% RSLogix 500 project BINSCRUBBER T SERIES WITH PALLET WASH AND STACKER_WITH_BIN_CALL_BAK721_eulises.RSS, saved by version 11.00.00.00 %
PROJECT "JBT BIN"    % processor: MicroLogix 1400 %

PROGRAM FILES
  LAD 2 "MAIN"  11 rungs
  LAD 3 "START_UP"  22 rungs
  LAD 4 "ENCODER"  11 rungs
  LAD 5 "CRADLE"  26 rungs
  LAD 6 "BRUSH"  53 rungs
  LAD 7 "TANK"  20 rungs
  LAD 8 "AUXILARY"  13 rungs
  LAD 9 "FAULTS"  37 rungs
  LAD 10 "PID ANALOG"  33 rungs  % Scaling %
  LAD 11 "BIN SIZING"  15 rungs  % Bin sizing Pallet, 26", Tall %
  LAD 12 "STACKER"  50 rungs

DATA FILES
  O0 OUTPUT  9 elements
  I1 INPUT  19 elements
  S2 STATUS  66 elements
  B3 BINARY  10 elements
  T4 TIMER  43 elements
  C5 COUNTER  1 elements
  R6 CONTROL  1 elements
  N7 INTEGER  62 elements
  F8 FLOAT  10 elements
  L9   1 elements
  L10   2 elements
  PD11   2 elements

LADDER 2 "MAIN"
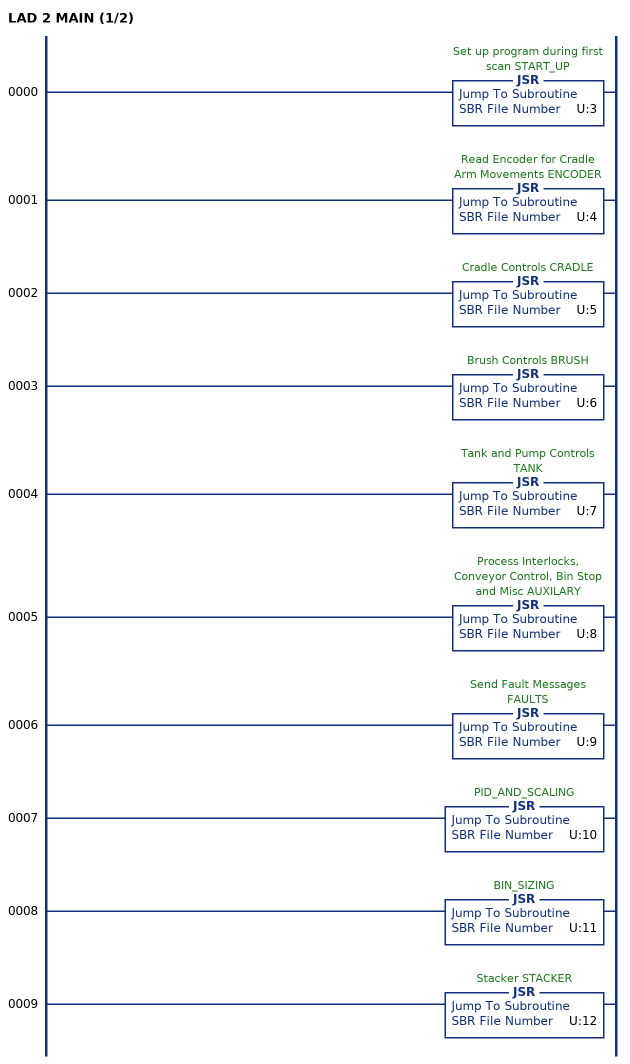
% Rung: 0 %
SOR JSR U:3 EOR
%   U:3  START_UP  "Set up program during first scan" %
% Rung: 1 %
SOR JSR U:4 EOR
%   U:4  ENCODER  "Read Encoder for Cradle Arm Movements" %
% Rung: 2 %
SOR JSR U:5 EOR
%   U:5  CRADLE  "Cradle Controls" %
% Rung: 3 %
SOR JSR U:6 EOR
%   U:6  BRUSH  "Brush Controls" %
% Rung: 4 %
SOR JSR U:7 EOR
%   U:7  TANK  "Tank and Pump Controls" %
% Rung: 5 %
SOR JSR U:8 EOR
%   U:8  AUXILARY  "Process Interlocks, Conveyor Control, Bin Stop and Misc" %
% Rung: 6 %
SOR JSR U:9 EOR
%   U:9  FAULTS  "Send Fault Messages" %
% Rung: 7 %
SOR JSR U:10 EOR
%   U:10  PID_AND_SCALING %
% Rung: 8 %
SOR JSR U:11 EOR
%   U:11  BIN_SIZING %
% Rung: 9 %
SOR JSR U:12 EOR
%   U:12  STACKER  "Stacker" %

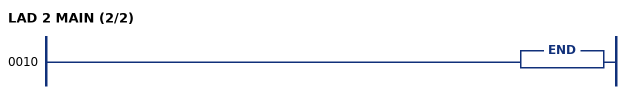
% Rung: 10 %
SOR END EOR

LADDER 3 "START_UP"
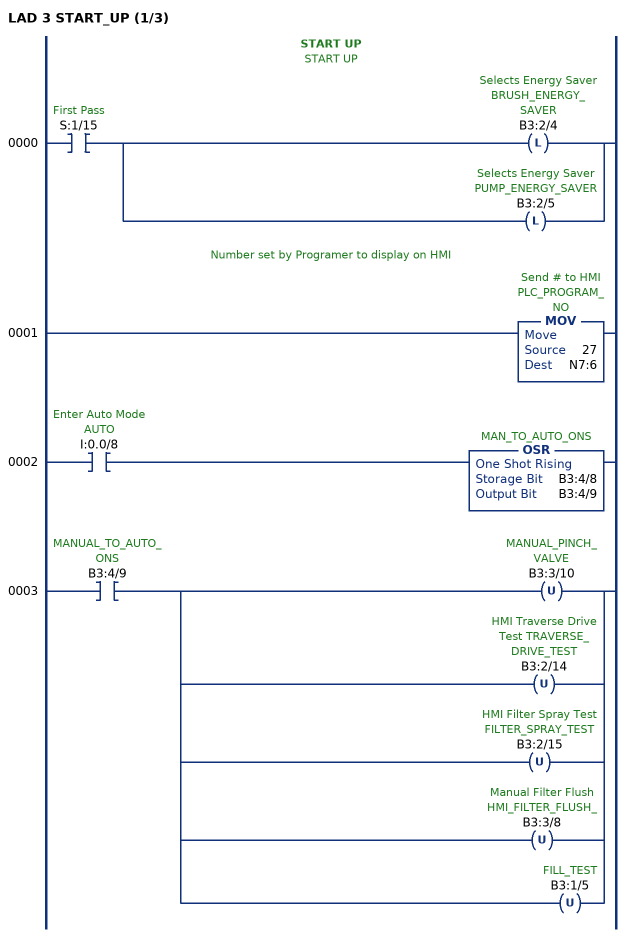
% Rung: 0 %
% TITLE: START UP %
% START UP %
SOR XIC S:1/15 BST OTL B3:2/4 NXB OTL B3:2/5 BND EOR
%   S:1/15  "First Pass" %
%   B3:2/4  BRUSH_ENERGY_SAVER  "Selects Energy Saver" %
%   B3:2/5  PUMP_ENERGY_SAVER  "Selects Energy Saver" %
% Rung: 1 %
% Number set by Programer to display on HMI %
SOR MOV 27 N7:6 EOR
%   N7:6  PLC_PROGRAM_NO  "Send # to HMI" %
% Rung: 2 %
SOR XIC I:0.0/8 OSR B3:4/8 B3:4/9 EOR
%   I:0.0/8  AUTO  "Enter Auto Mode" %
%   B3:4/8  MAN_TO_AUTO_ONS %
%   B3:4/9  MANUAL_TO_AUTO_ONS %
% Rung: 3 %
SOR XIC B3:4/9 BST OTU B3:3/10 NXB BST OTU B3:2/14 NXB BST OTU B3:2/15 NXB BST OTU B3:3/8 NXB OTU B3:1/5 BND BND BND BND EOR
%   B3:4/9  MANUAL_TO_AUTO_ONS %
%   B3:3/10  MANUAL_PINCH_VALVE %
%   B3:2/14  TRAVERSE_DRIVE_TEST  "HMI Traverse Drive Test" %
%   B3:2/15  FILTER_SPRAY_TEST  "HMI Filter Spray Test" %
%   B3:3/8  HMI_FILTER_FLUSH_  "Manual Filter Flush" %
%   B3:1/5  FILL_TEST %

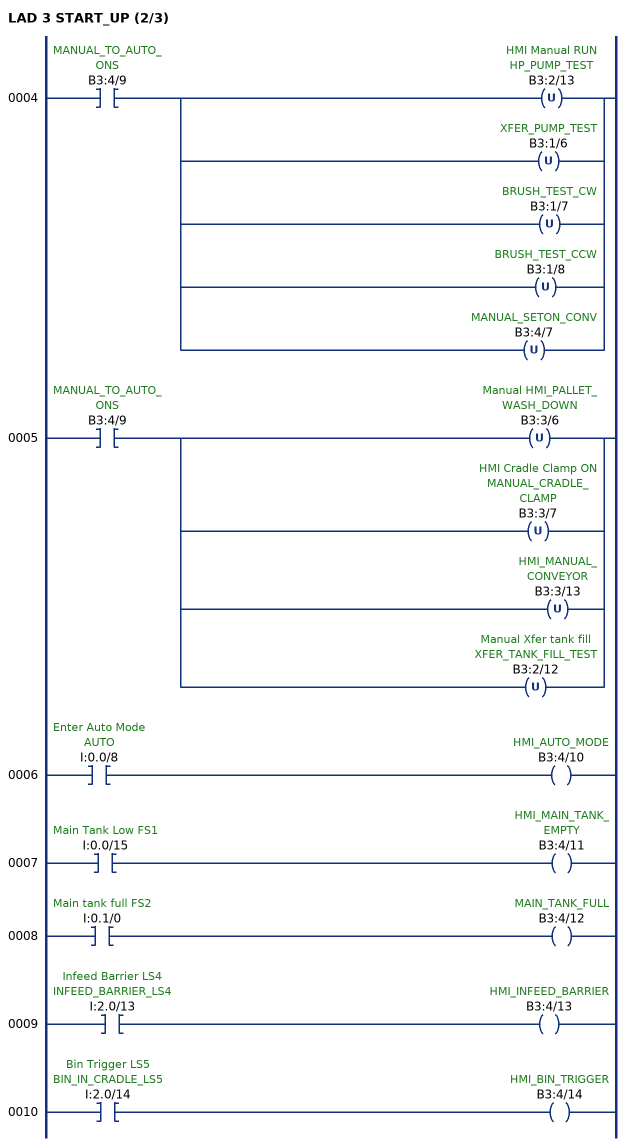
% Rung: 4 %
SOR XIC B3:4/9 BST OTU B3:2/13 NXB BST OTU B3:1/6 NXB BST OTU B3:1/7 NXB BST OTU B3:1/8 NXB OTU B3:4/7 BND BND BND BND EOR
%   B3:4/9  MANUAL_TO_AUTO_ONS %
%   B3:2/13  HP_PUMP_TEST  "HMI Manual RUN" %
%   B3:1/6  XFER_PUMP_TEST %
%   B3:1/7  BRUSH_TEST_CW %
%   B3:1/8  BRUSH_TEST_CCW %
%   B3:4/7  MANUAL_SETON_CONV %
% Rung: 5 %
SOR XIC B3:4/9 BST OTU B3:3/6 NXB BST OTU B3:3/7 NXB BST OTU B3:3/13 NXB OTU B3:2/12 BND BND BND EOR
%   B3:4/9  MANUAL_TO_AUTO_ONS %
%   B3:3/6  HMI_PALLET_WASH_DOWN  "Manual" %
%   B3:3/7  MANUAL_CRADLE_CLAMP  "HMI Cradle Clamp ON" %
%   B3:3/13  HMI_MANUAL_CONVEYOR %
%   B3:2/12  XFER_TANK_FILL_TEST  "Manual Xfer tank fill" %
% Rung: 6 %
SOR XIC I:0.0/8 OTE B3:4/10 EOR
%   I:0.0/8  AUTO  "Enter Auto Mode" %
%   B3:4/10  HMI_AUTO_MODE %
% Rung: 7 %
SOR XIC I:0.0/15 OTE B3:4/11 EOR
%   I:0.0/15  FS1  "Main Tank Low" %
%   B3:4/11  HMI_MAIN_TANK_EMPTY %
% Rung: 8 %
SOR XIC I:0.1/0 OTE B3:4/12 EOR
%   I:0.1/0  FS2  "Main tank full" %
%   B3:4/12  MAIN_TANK_FULL %
% Rung: 9 %
SOR XIC I:2.0/13 OTE B3:4/13 EOR
%   I:2.0/13  INFEED_BARRIER_LS4  "Infeed Barrier LS4" %
%   B3:4/13  HMI_INFEED_BARRIER %
% Rung: 10 %
SOR XIC I:2.0/14 OTE B3:4/14 EOR
%   I:2.0/14  BIN_IN_CRADLE_LS5  "Bin Trigger LS5" %
%   B3:4/14  HMI_BIN_TRIGGER %

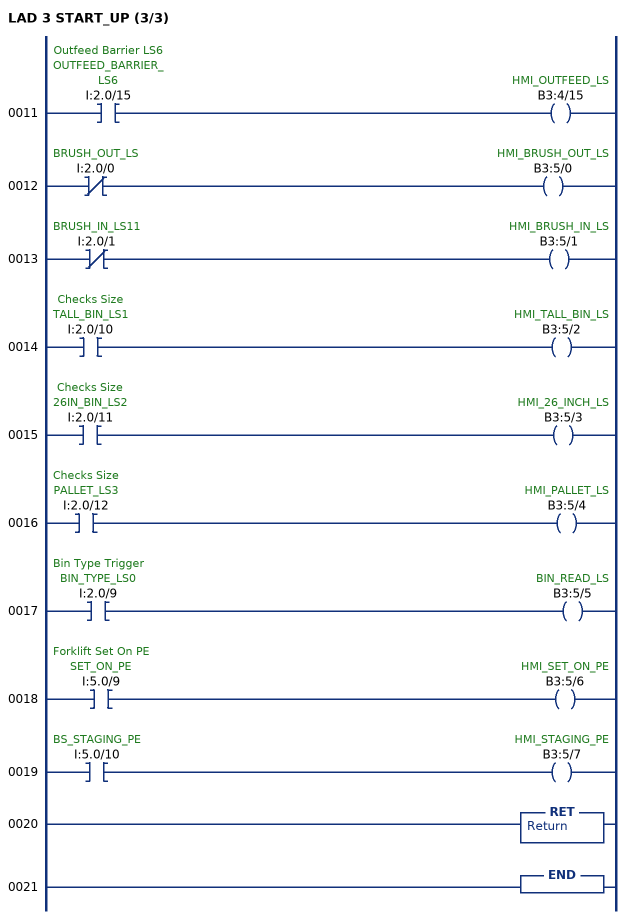
% Rung: 11 %
SOR XIC I:2.0/15 OTE B3:4/15 EOR
%   I:2.0/15  OUTFEED_BARRIER_LS6  "Outfeed Barrier LS6" %
%   B3:4/15  HMI_OUTFEED_LS %
% Rung: 12 %
SOR XIO I:2.0/0 OTE B3:5/0 EOR
%   I:2.0/0  BRUSH_OUT_LS %
%   B3:5/0  HMI_BRUSH_OUT_LS %
% Rung: 13 %
SOR XIO I:2.0/1 OTE B3:5/1 EOR
%   I:2.0/1  BRUSH_IN_LS11 %
%   B3:5/1  HMI_BRUSH_IN_LS %
% Rung: 14 %
SOR XIC I:2.0/10 OTE B3:5/2 EOR
%   I:2.0/10  TALL_BIN_LS1  "Checks Size" %
%   B3:5/2  HMI_TALL_BIN_LS %
% Rung: 15 %
SOR XIC I:2.0/11 OTE B3:5/3 EOR
%   I:2.0/11  26IN_BIN_LS2  "Checks Size" %
%   B3:5/3  HMI_26_INCH_LS %
% Rung: 16 %
SOR XIC I:2.0/12 OTE B3:5/4 EOR
%   I:2.0/12  PALLET_LS3  "Checks Size" %
%   B3:5/4  HMI_PALLET_LS %
% Rung: 17 %
SOR XIC I:2.0/9 OTE B3:5/5 EOR
%   I:2.0/9  BIN_TYPE_LS0  "Bin Type Trigger" %
%   B3:5/5  BIN_READ_LS %
% Rung: 18 %
SOR XIC I:5.0/9 OTE B3:5/6 EOR
%   I:5.0/9  SET_ON_PE  "Forklift Set On PE" %
%   B3:5/6  HMI_SET_ON_PE %
% Rung: 19 %
SOR XIC I:5.0/10 OTE B3:5/7 EOR
%   I:5.0/10  BS_STAGING_PE %
%   B3:5/7  HMI_STAGING_PE %
% Rung: 20 %
SOR RET EOR
% Rung: 21 %
SOR END EOR

LADDER 4 "ENCODER"
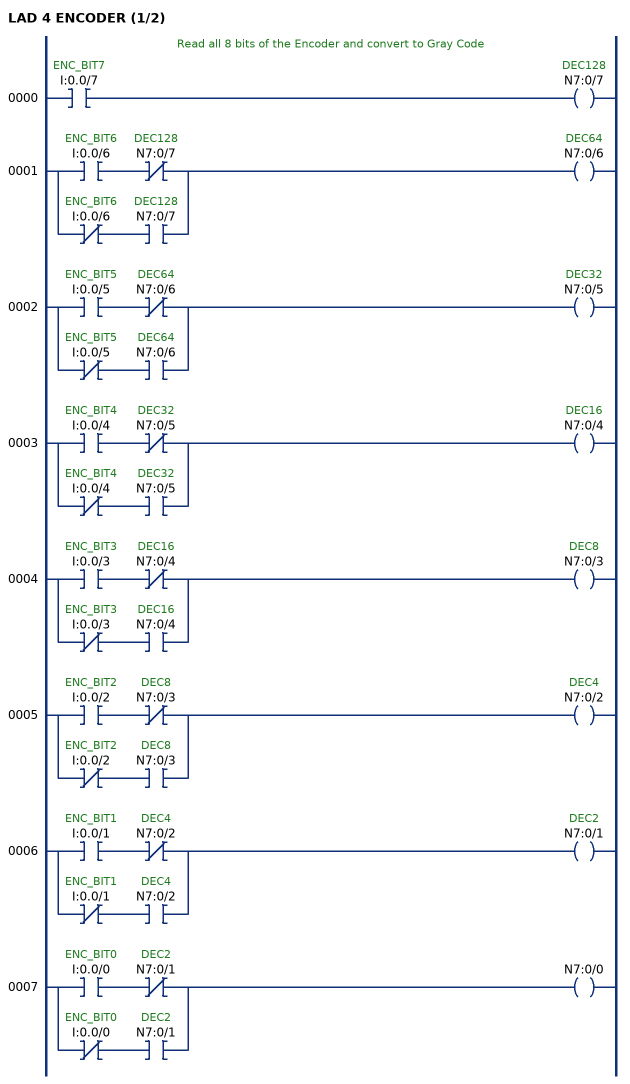
% Rung: 0 %
% Read all 8 bits of the Encoder and convert to Gray Code %
SOR XIC I:0.0/7 OTE N7:0/7 EOR
%   I:0.0/7  ENC_BIT7 %
%   N7:0/7  "DEC128" %
% Rung: 1 %
SOR BST XIC I:0.0/6 XIO N7:0/7 NXB XIO I:0.0/6 XIC N7:0/7 BND OTE N7:0/6 EOR
%   I:0.0/6  ENC_BIT6 %
%   N7:0/7  "DEC128" %
%   N7:0/6  "DEC64" %
% Rung: 2 %
SOR BST XIC I:0.0/5 XIO N7:0/6 NXB XIO I:0.0/5 XIC N7:0/6 BND OTE N7:0/5 EOR
%   I:0.0/5  ENC_BIT5 %
%   N7:0/6  "DEC64" %
%   N7:0/5  "DEC32" %
% Rung: 3 %
SOR BST XIC I:0.0/4 XIO N7:0/5 NXB XIO I:0.0/4 XIC N7:0/5 BND OTE N7:0/4 EOR
%   I:0.0/4  ENC_BIT4 %
%   N7:0/5  "DEC32" %
%   N7:0/4  "DEC16" %
% Rung: 4 %
SOR BST XIC I:0.0/3 XIO N7:0/4 NXB XIO I:0.0/3 XIC N7:0/4 BND OTE N7:0/3 EOR
%   I:0.0/3  ENC_BIT3 %
%   N7:0/4  "DEC16" %
%   N7:0/3  "DEC8" %
% Rung: 5 %
SOR BST XIC I:0.0/2 XIO N7:0/3 NXB XIO I:0.0/2 XIC N7:0/3 BND OTE N7:0/2 EOR
%   I:0.0/2  ENC_BIT2 %
%   N7:0/3  "DEC8" %
%   N7:0/2  "DEC4" %
% Rung: 6 %
SOR BST XIC I:0.0/1 XIO N7:0/2 NXB XIO I:0.0/1 XIC N7:0/2 BND OTE N7:0/1 EOR
%   I:0.0/1  ENC_BIT1 %
%   N7:0/2  "DEC4" %
%   N7:0/1  "DEC2" %
% Rung: 7 %
SOR BST XIC I:0.0/0 XIO N7:0/1 NXB XIO I:0.0/0 XIC N7:0/1 BND OTE N7:0/0 EOR
%   I:0.0/0  ENC_BIT0 %
%   N7:0/1  "DEC2" %

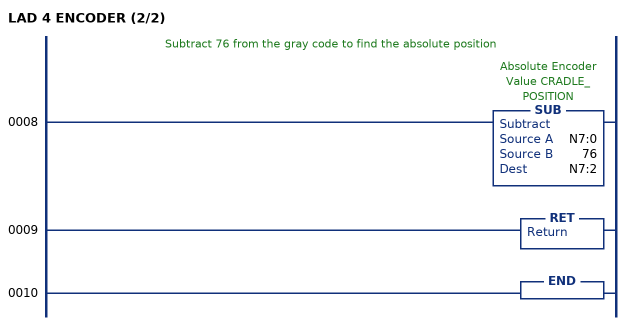
% Rung: 8 %
% Subtract 76 from the gray code to find the absolute position %
SOR SUB N7:0 76 N7:2 EOR
%   N7:0  ENC_POS %
%   N7:2  CRADLE_POSITION  "Absolute Encoder Value" %
% Rung: 9 %
SOR RET EOR
% Rung: 10 %
SOR END EOR

LADDER 5 "CRADLE"
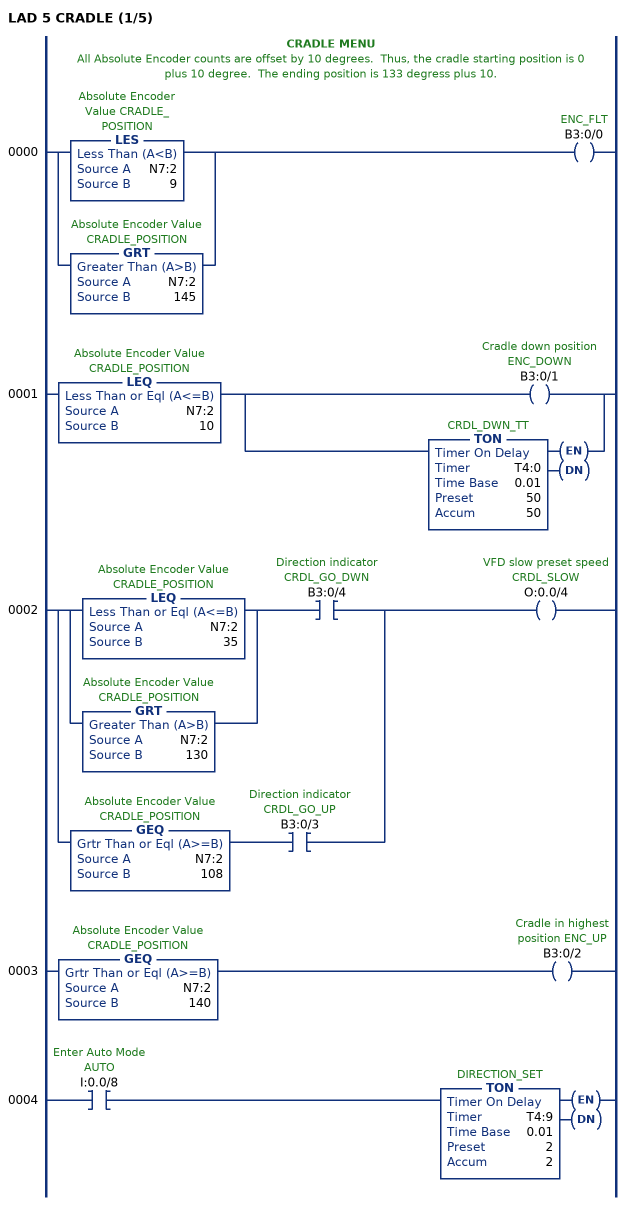
% Rung: 0 %
% TITLE: CRADLE MENU %
% All Absolute Encoder counts are offset by 10 degrees.  Thus, the cradle starting position is 0 plus 10 degree.  The ending position is 133 degress plus 10. %
SOR BST LES N7:2 9 NXB GRT N7:2 145 BND OTE B3:0/0 EOR
%   N7:2  CRADLE_POSITION  "Absolute Encoder Value" %
%   B3:0/0  ENC_FLT %
% Rung: 1 %
SOR LEQ N7:2 10 BST OTE B3:0/1 NXB TON T4:0 0.01 50 50 BND EOR
%   N7:2  CRADLE_POSITION  "Absolute Encoder Value" %
%   B3:0/1  ENC_DOWN  "Cradle down position" %
%   T4:0  CRDL_DWN_TT %
% Rung: 2 %
SOR BST BST LEQ N7:2 35 NXB GRT N7:2 130 BND XIC B3:0/4 NXB GEQ N7:2 108 XIC B3:0/3 BND OTE O:0.0/4 EOR
%   N7:2  CRADLE_POSITION  "Absolute Encoder Value" %
%   B3:0/4  CRDL_GO_DWN  "Direction indicator" %
%   B3:0/3  CRDL_GO_UP  "Direction indicator" %
%   O:0.0/4  CRDL_SLOW  "VFD slow preset speed" %
% Rung: 3 %
SOR GEQ N7:2 140 OTE B3:0/2 EOR
%   N7:2  CRADLE_POSITION  "Absolute Encoder Value" %
%   B3:0/2  ENC_UP  "Cradle in highest position" %
% Rung: 4 %
SOR XIC I:0.0/8 TON T4:9 0.01 2 2 EOR
%   I:0.0/8  AUTO  "Enter Auto Mode" %
%   T4:9  DIRECTION_SET %

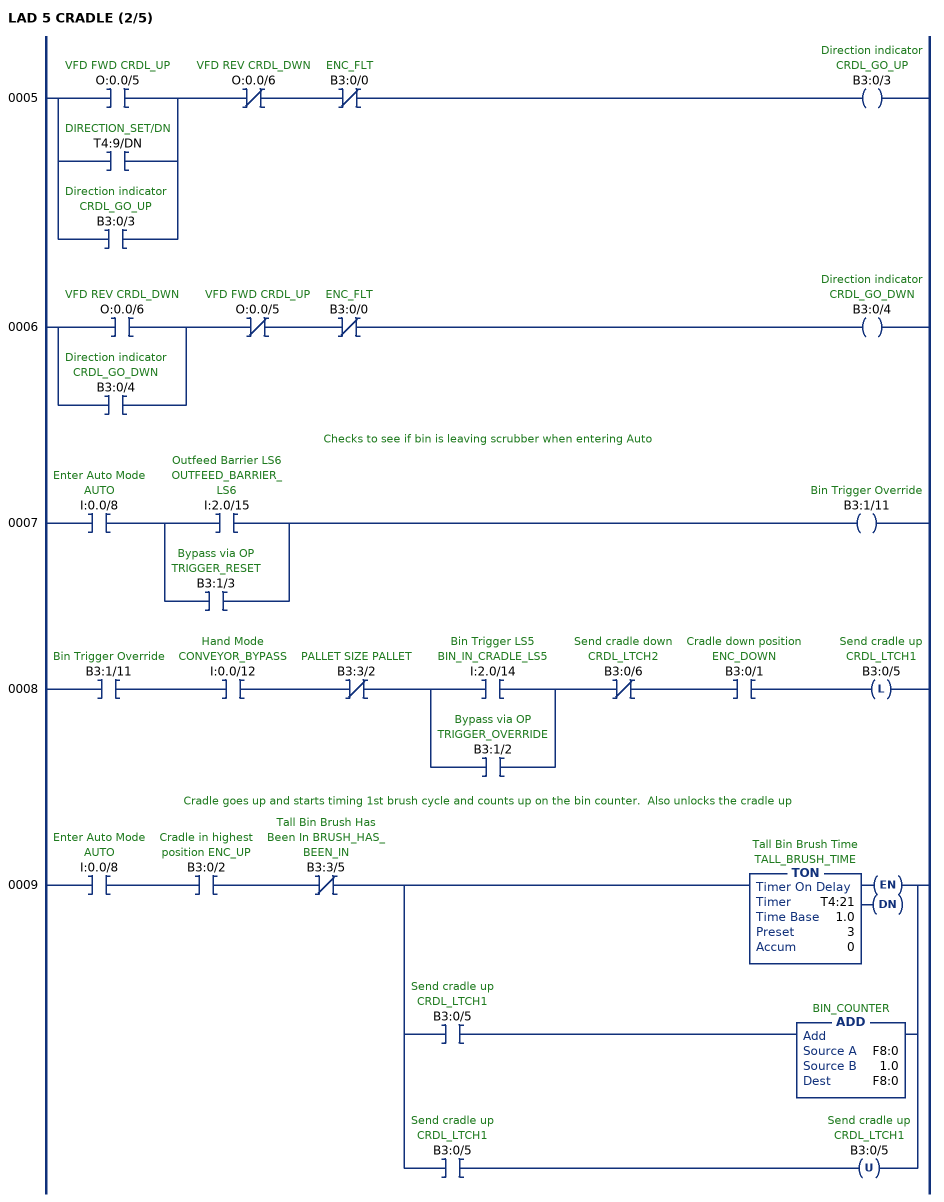
% Rung: 5 %
SOR BST XIC O:0.0/5 NXB XIC T4:9/DN NXB XIC B3:0/3 BND XIO O:0.0/6 XIO B3:0/0 OTE B3:0/3 EOR
%   O:0.0/5  CRDL_UP  "VFD FWD" %
%   T4:9  DIRECTION_SET %
%   B3:0/3  CRDL_GO_UP  "Direction indicator" %
%   O:0.0/6  CRDL_DWN  "VFD REV" %
%   B3:0/0  ENC_FLT %
% Rung: 6 %
SOR BST XIC O:0.0/6 NXB XIC B3:0/4 BND XIO O:0.0/5 XIO B3:0/0 OTE B3:0/4 EOR
%   O:0.0/6  CRDL_DWN  "VFD REV" %
%   B3:0/4  CRDL_GO_DWN  "Direction indicator" %
%   O:0.0/5  CRDL_UP  "VFD FWD" %
%   B3:0/0  ENC_FLT %
% Rung: 7 %
% Checks to see if bin is leaving scrubber when entering Auto %
SOR XIC I:0.0/8 BST XIC I:2.0/15 NXB XIC B3:1/3 BND OTE B3:1/11 EOR
%   I:0.0/8  AUTO  "Enter Auto Mode" %
%   I:2.0/15  OUTFEED_BARRIER_LS6  "Outfeed Barrier LS6" %
%   B3:1/3  TRIGGER_RESET  "Bypass via OP" %
%   B3:1/11  "Bin Trigger Override" %
% Rung: 8 %
SOR XIC B3:1/11 XIC I:0.0/12 XIO B3:3/2 BST XIC I:2.0/14 NXB XIC B3:1/2 BND XIO B3:0/6 XIC B3:0/1 OTL B3:0/5 EOR
%   B3:1/11  "Bin Trigger Override" %
%   I:0.0/12  CONVEYOR_BYPASS  "Hand Mode" %
%   B3:3/2  PALLET  "PALLET SIZE" %
%   I:2.0/14  BIN_IN_CRADLE_LS5  "Bin Trigger LS5" %
%   B3:1/2  TRIGGER_OVERRIDE  "Bypass via OP" %
%   B3:0/6  CRDL_LTCH2  "Send cradle down" %
%   B3:0/1  ENC_DOWN  "Cradle down position" %
%   B3:0/5  CRDL_LTCH1  "Send cradle up" %
% Rung: 9 %
% Cradle goes up and starts timing 1st brush cycle and counts up on the bin counter.  Also unlocks the cradle up %
SOR XIC I:0.0/8 XIC B3:0/2 XIO B3:3/5 BST TON T4:21 1.0 3 0 NXB BST XIC B3:0/5 ADD F8:0 1.0 F8:0 NXB XIC B3:0/5 OTU B3:0/5 BND BND EOR
%   I:0.0/8  AUTO  "Enter Auto Mode" %
%   B3:0/2  ENC_UP  "Cradle in highest position" %
%   B3:3/5  BRUSH_HAS_BEEN_IN  "Tall Bin Brush Has Been In" %
%   T4:21  TALL_BRUSH_TIME  "Tall Bin Brush Time" %
%   B3:0/5  CRDL_LTCH1  "Send cradle up" %
%   F8:0  BIN_COUNTER %

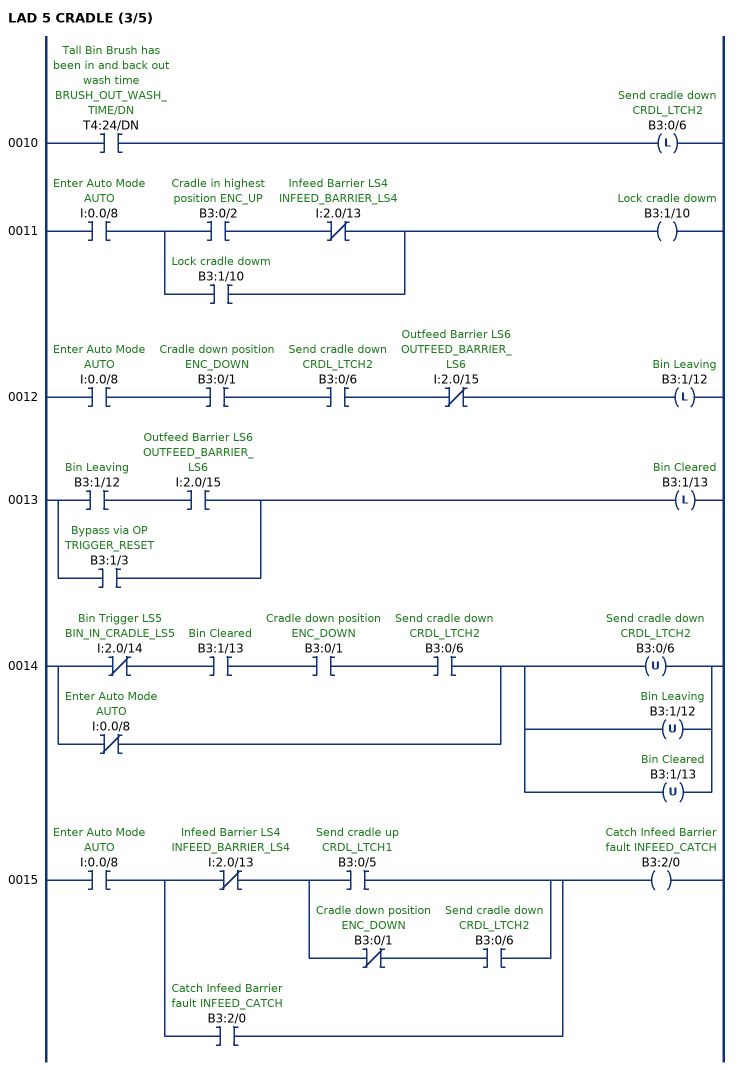
% Rung: 10 %
SOR XIC T4:24/DN OTL B3:0/6 EOR
%   T4:24  BRUSH_OUT_WASH_TIME  "Tall Bin Brush has been in and back out wash time" %
%   B3:0/6  CRDL_LTCH2  "Send cradle down" %
% Rung: 11 %
SOR XIC I:0.0/8 BST XIC B3:0/2 XIO I:2.0/13 NXB XIC B3:1/10 BND OTE B3:1/10 EOR
%   I:0.0/8  AUTO  "Enter Auto Mode" %
%   B3:0/2  ENC_UP  "Cradle in highest position" %
%   I:2.0/13  INFEED_BARRIER_LS4  "Infeed Barrier LS4" %
%   B3:1/10  "Lock cradle dowm" %
% Rung: 12 %
SOR XIC I:0.0/8 XIC B3:0/1 XIC B3:0/6 XIO I:2.0/15 OTL B3:1/12 EOR
%   I:0.0/8  AUTO  "Enter Auto Mode" %
%   B3:0/1  ENC_DOWN  "Cradle down position" %
%   B3:0/6  CRDL_LTCH2  "Send cradle down" %
%   I:2.0/15  OUTFEED_BARRIER_LS6  "Outfeed Barrier LS6" %
%   B3:1/12  "Bin Leaving" %
% Rung: 13 %
SOR BST XIC B3:1/12 XIC I:2.0/15 NXB XIC B3:1/3 BND OTL B3:1/13 EOR
%   B3:1/12  "Bin Leaving" %
%   I:2.0/15  OUTFEED_BARRIER_LS6  "Outfeed Barrier LS6" %
%   B3:1/3  TRIGGER_RESET  "Bypass via OP" %
%   B3:1/13  "Bin Cleared" %
% Rung: 14 %
SOR BST XIO I:2.0/14 XIC B3:1/13 XIC B3:0/1 XIC B3:0/6 NXB XIO I:0.0/8 BND BST OTU B3:0/6 NXB BST OTU B3:1/12 NXB OTU B3:1/13 BND BND EOR
%   I:2.0/14  BIN_IN_CRADLE_LS5  "Bin Trigger LS5" %
%   B3:1/13  "Bin Cleared" %
%   B3:0/1  ENC_DOWN  "Cradle down position" %
%   B3:0/6  CRDL_LTCH2  "Send cradle down" %
%   I:0.0/8  AUTO  "Enter Auto Mode" %
%   B3:1/12  "Bin Leaving" %
% Rung: 15 %
SOR XIC I:0.0/8 BST XIO I:2.0/13 BST XIC B3:0/5 NXB XIO B3:0/1 XIC B3:0/6 BND NXB XIC B3:2/0 BND OTE B3:2/0 EOR
%   I:0.0/8  AUTO  "Enter Auto Mode" %
%   I:2.0/13  INFEED_BARRIER_LS4  "Infeed Barrier LS4" %
%   B3:0/5  CRDL_LTCH1  "Send cradle up" %
%   B3:0/1  ENC_DOWN  "Cradle down position" %
%   B3:0/6  CRDL_LTCH2  "Send cradle down" %
%   B3:2/0  INFEED_CATCH  "Catch Infeed Barrier fault" %

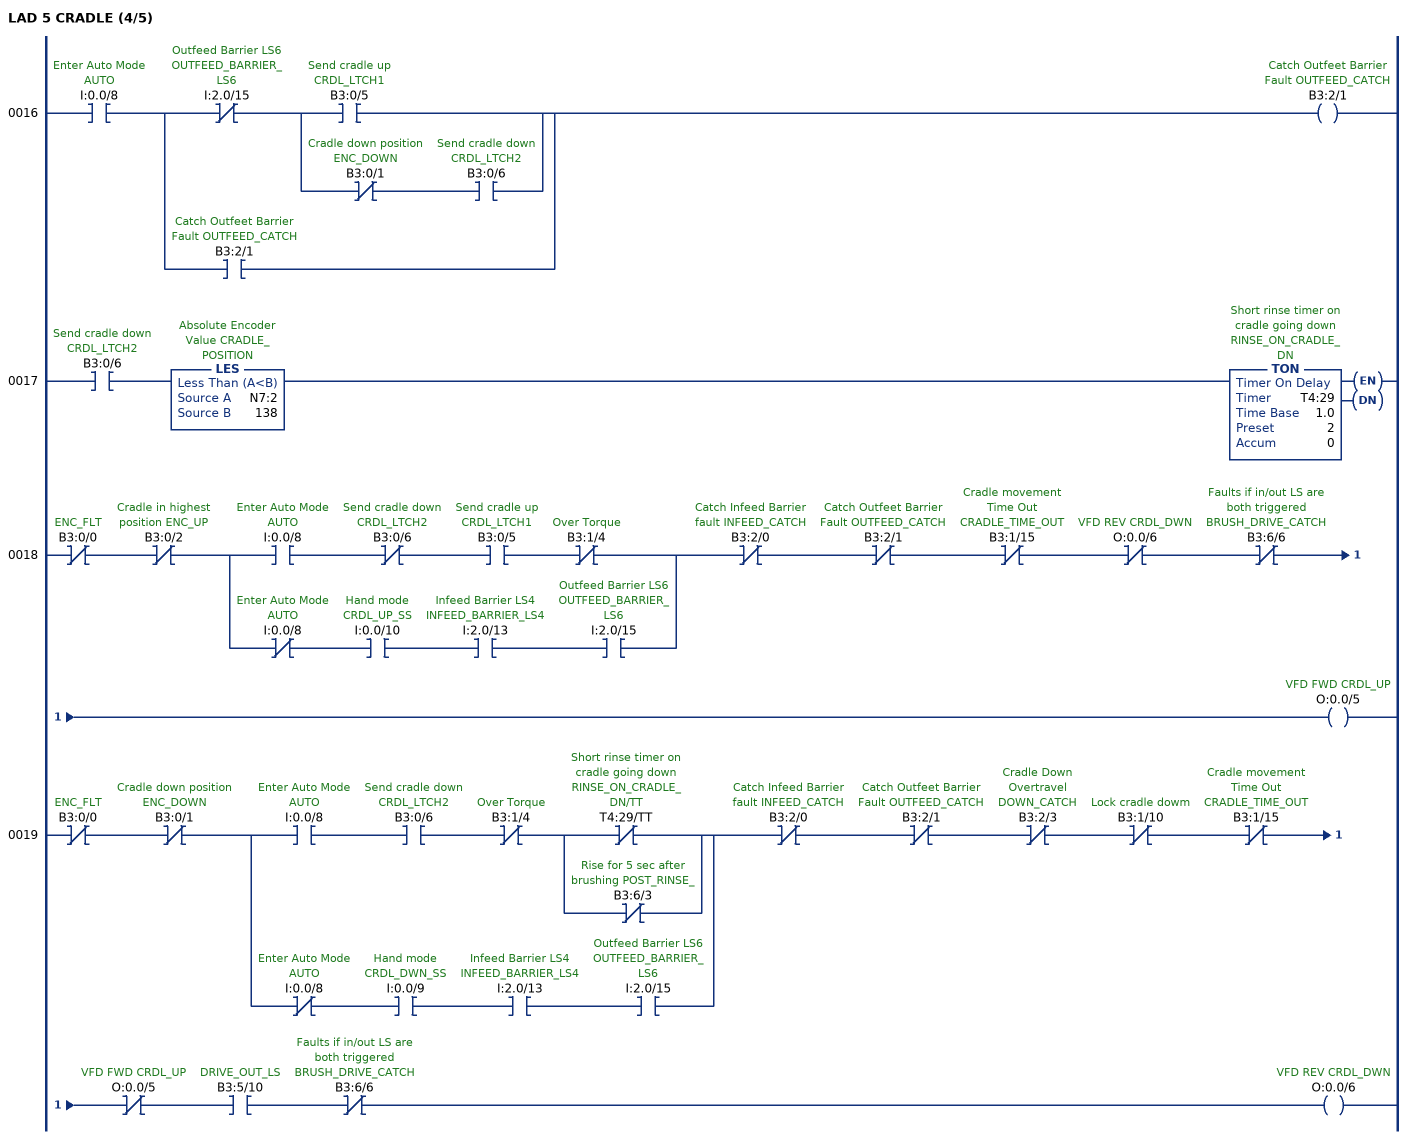
% Rung: 16 %
SOR XIC I:0.0/8 BST XIO I:2.0/15 BST XIC B3:0/5 NXB XIO B3:0/1 XIC B3:0/6 BND NXB XIC B3:2/1 BND OTE B3:2/1 EOR
%   I:0.0/8  AUTO  "Enter Auto Mode" %
%   I:2.0/15  OUTFEED_BARRIER_LS6  "Outfeed Barrier LS6" %
%   B3:0/5  CRDL_LTCH1  "Send cradle up" %
%   B3:0/1  ENC_DOWN  "Cradle down position" %
%   B3:0/6  CRDL_LTCH2  "Send cradle down" %
%   B3:2/1  OUTFEED_CATCH  "Catch Outfeet Barrier Fault" %
% Rung: 17 %
SOR XIC B3:0/6 LES N7:2 138 TON T4:29 1.0 2 0 EOR
%   B3:0/6  CRDL_LTCH2  "Send cradle down" %
%   N7:2  CRADLE_POSITION  "Absolute Encoder Value" %
%   T4:29  RINSE_ON_CRADLE_DN  "Short rinse timer on cradle going down" %
% Rung: 18 %
SOR XIO B3:0/0 XIO B3:0/2 BST XIC I:0.0/8 XIO B3:0/6 XIC B3:0/5 XIO B3:1/4 NXB XIO I:0.0/8 XIC I:0.0/10 XIC I:2.0/13 XIC I:2.0/15 BND XIO B3:2/0 XIO B3:2/1 XIO B3:1/15 XIO O:0.0/6 XIO B3:6/6 OTE O:0.0/5 EOR
%   B3:0/0  ENC_FLT %
%   B3:0/2  ENC_UP  "Cradle in highest position" %
%   I:0.0/8  AUTO  "Enter Auto Mode" %
%   B3:0/6  CRDL_LTCH2  "Send cradle down" %
%   B3:0/5  CRDL_LTCH1  "Send cradle up" %
%   B3:1/4  "Over Torque" %
%   I:0.0/10  CRDL_UP_SS  "Hand mode" %
%   I:2.0/13  INFEED_BARRIER_LS4  "Infeed Barrier LS4" %
%   I:2.0/15  OUTFEED_BARRIER_LS6  "Outfeed Barrier LS6" %
%   B3:2/0  INFEED_CATCH  "Catch Infeed Barrier fault" %
%   B3:2/1  OUTFEED_CATCH  "Catch Outfeet Barrier Fault" %
%   B3:1/15  CRADLE_TIME_OUT  "Cradle movement Time Out" %
%   O:0.0/6  CRDL_DWN  "VFD REV" %
%   B3:6/6  BRUSH_DRIVE_CATCH  "Faults if in/out LS are both triggered" %
%   O:0.0/5  CRDL_UP  "VFD FWD" %
% Rung: 19 %
SOR XIO B3:0/0 XIO B3:0/1 BST XIC I:0.0/8 XIC B3:0/6 XIO B3:1/4 BST XIO T4:29/TT NXB XIO B3:6/3 BND NXB XIO I:0.0/8 XIC I:0.0/9 XIC I:2.0/13 XIC I:2.0/15 BND XIO B3:2/0 XIO B3:2/1 XIO B3:2/3 XIO B3:1/10 XIO B3:1/15 XIO O:0.0/5 XIC B3:5/10 XIO B3:6/6 OTE O:0.0/6 EOR
%   B3:0/0  ENC_FLT %
%   B3:0/1  ENC_DOWN  "Cradle down position" %
%   I:0.0/8  AUTO  "Enter Auto Mode" %
%   B3:0/6  CRDL_LTCH2  "Send cradle down" %
%   B3:1/4  "Over Torque" %
%   T4:29  RINSE_ON_CRADLE_DN  "Short rinse timer on cradle going down" %
%   B3:6/3  POST_RINSE_  "Rise for 5 sec after brushing" %
%   I:0.0/9  CRDL_DWN_SS  "Hand mode" %
%   I:2.0/13  INFEED_BARRIER_LS4  "Infeed Barrier LS4" %
%   I:2.0/15  OUTFEED_BARRIER_LS6  "Outfeed Barrier LS6" %
%   B3:2/0  INFEED_CATCH  "Catch Infeed Barrier fault" %
%   B3:2/1  OUTFEED_CATCH  "Catch Outfeet Barrier Fault" %
%   B3:2/3  DOWN_CATCH  "Cradle Down Overtravel" %
%   B3:1/10  "Lock cradle dowm" %
%   B3:1/15  CRADLE_TIME_OUT  "Cradle movement Time Out" %
%   O:0.0/5  CRDL_UP  "VFD FWD" %
%   B3:5/10  DRIVE_OUT_LS %
%   B3:6/6  BRUSH_DRIVE_CATCH  "Faults if in/out LS are both triggered" %
%   O:0.0/6  CRDL_DWN  "VFD REV" %

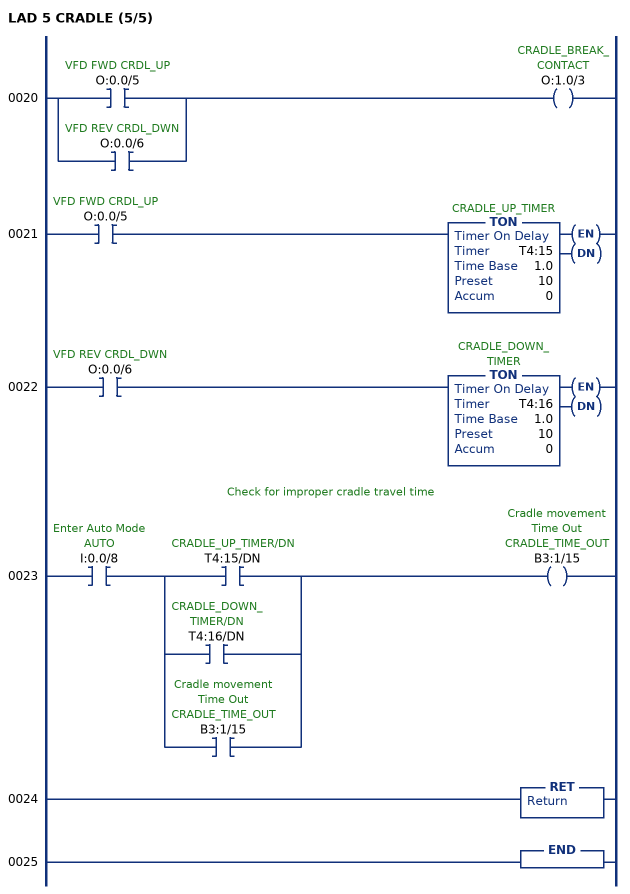
% Rung: 20 %
SOR BST XIC O:0.0/5 NXB XIC O:0.0/6 BND OTE O:1.0/3 EOR
%   O:0.0/5  CRDL_UP  "VFD FWD" %
%   O:0.0/6  CRDL_DWN  "VFD REV" %
%   O:1.0/3  CRADLE_BREAK_CONTACT %
% Rung: 21 %
SOR XIC O:0.0/5 TON T4:15 1.0 10 0 EOR
%   O:0.0/5  CRDL_UP  "VFD FWD" %
%   T4:15  CRADLE_UP_TIMER %
% Rung: 22 %
SOR XIC O:0.0/6 TON T4:16 1.0 10 0 EOR
%   O:0.0/6  CRDL_DWN  "VFD REV" %
%   T4:16  CRADLE_DOWN_TIMER %
% Rung: 23 %
% Check for improper cradle travel time %
SOR XIC I:0.0/8 BST BST XIC T4:15/DN NXB XIC T4:16/DN BND NXB XIC B3:1/15 BND OTE B3:1/15 EOR
%   I:0.0/8  AUTO  "Enter Auto Mode" %
%   T4:15  CRADLE_UP_TIMER %
%   T4:16  CRADLE_DOWN_TIMER %
%   B3:1/15  CRADLE_TIME_OUT  "Cradle movement Time Out" %
% Rung: 24 %
SOR RET EOR
% Rung: 25 %
SOR END EOR

LADDER 6 "BRUSH"
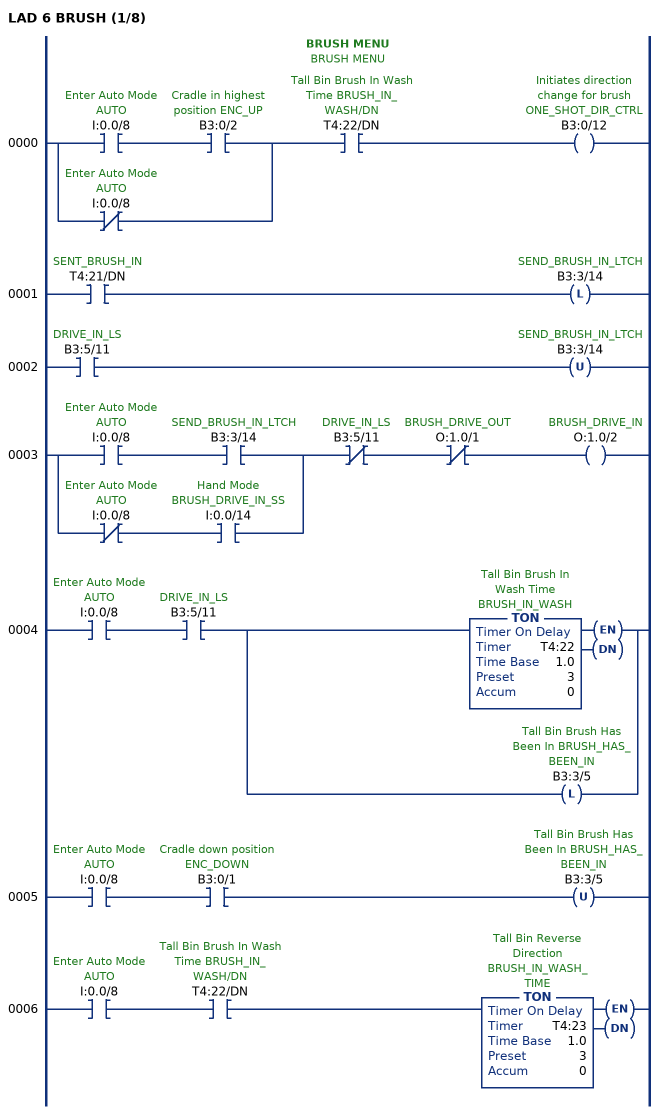
% Rung: 0 %
% TITLE: BRUSH MENU %
% BRUSH MENU %
SOR BST XIC I:0.0/8 XIC B3:0/2 NXB XIO I:0.0/8 BND XIC T4:22/DN OTE B3:0/12 EOR
%   I:0.0/8  AUTO  "Enter Auto Mode" %
%   B3:0/2  ENC_UP  "Cradle in highest position" %
%   T4:22  BRUSH_IN_WASH  "Tall Bin Brush In Wash Time" %
%   B3:0/12  ONE_SHOT_DIR_CTRL  "Initiates direction change for brush" %
% Rung: 1 %
SOR XIC T4:21/DN OTL B3:3/14 EOR
%   T4:21/DN  SENT_BRUSH_IN %
%   B3:3/14  SEND_BRUSH_IN_LTCH %
% Rung: 2 %
SOR XIC B3:5/11 OTU B3:3/14 EOR
%   B3:5/11  DRIVE_IN_LS %
%   B3:3/14  SEND_BRUSH_IN_LTCH %
% Rung: 3 %
SOR BST XIC I:0.0/8 XIC B3:3/14 NXB XIO I:0.0/8 XIC I:0.0/14 BND XIO B3:5/11 XIO O:1.0/1 OTE O:1.0/2 EOR
%   I:0.0/8  AUTO  "Enter Auto Mode" %
%   B3:3/14  SEND_BRUSH_IN_LTCH %
%   I:0.0/14  BRUSH_DRIVE_IN_SS  "Hand Mode" %
%   B3:5/11  DRIVE_IN_LS %
%   O:1.0/1  BRUSH_DRIVE_OUT %
%   O:1.0/2  BRUSH_DRIVE_IN %
% Rung: 4 %
SOR XIC I:0.0/8 XIC B3:5/11 BST TON T4:22 1.0 3 0 NXB OTL B3:3/5 BND EOR
%   I:0.0/8  AUTO  "Enter Auto Mode" %
%   B3:5/11  DRIVE_IN_LS %
%   T4:22  BRUSH_IN_WASH  "Tall Bin Brush In Wash Time" %
%   B3:3/5  BRUSH_HAS_BEEN_IN  "Tall Bin Brush Has Been In" %
% Rung: 5 %
SOR XIC I:0.0/8 XIC B3:0/1 OTU B3:3/5 EOR
%   I:0.0/8  AUTO  "Enter Auto Mode" %
%   B3:0/1  ENC_DOWN  "Cradle down position" %
%   B3:3/5  BRUSH_HAS_BEEN_IN  "Tall Bin Brush Has Been In" %
% Rung: 6 %
SOR XIC I:0.0/8 XIC T4:22/DN TON T4:23 1.0 3 0 EOR
%   I:0.0/8  AUTO  "Enter Auto Mode" %
%   T4:22  BRUSH_IN_WASH  "Tall Bin Brush In Wash Time" %
%   T4:23  BRUSH_IN_WASH_TIME  "Tall Bin Reverse Direction" %

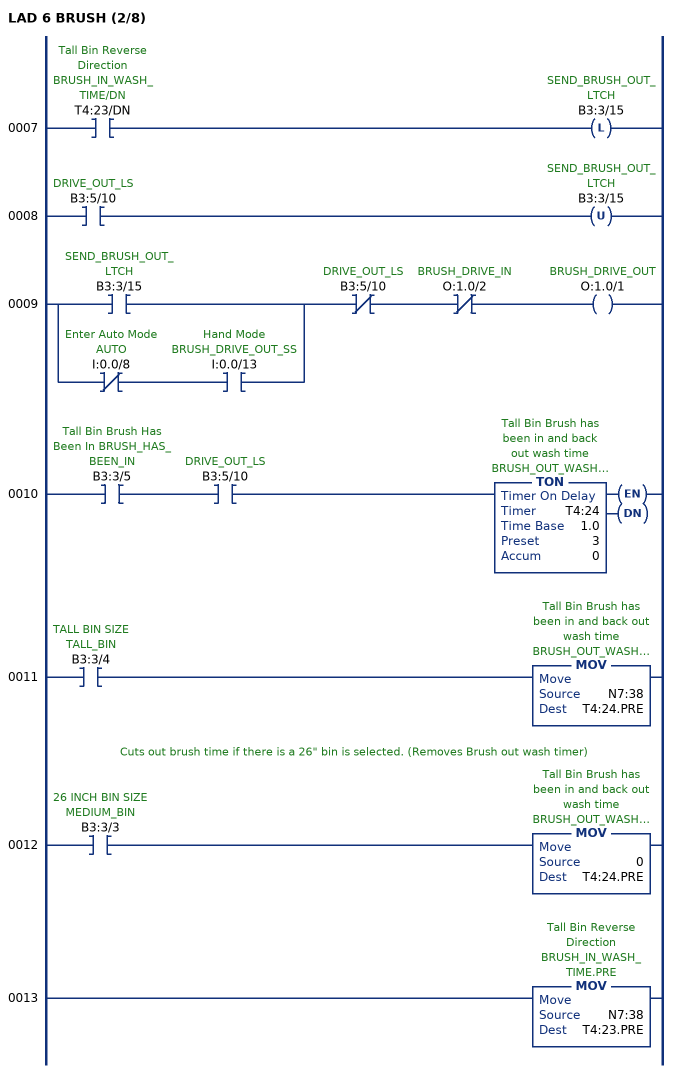
% Rung: 7 %
SOR XIC T4:23/DN OTL B3:3/15 EOR
%   T4:23  BRUSH_IN_WASH_TIME  "Tall Bin Reverse Direction" %
%   B3:3/15  SEND_BRUSH_OUT_LTCH %
% Rung: 8 %
SOR XIC B3:5/10 OTU B3:3/15 EOR
%   B3:5/10  DRIVE_OUT_LS %
%   B3:3/15  SEND_BRUSH_OUT_LTCH %
% Rung: 9 %
SOR BST XIC B3:3/15 NXB XIO I:0.0/8 XIC I:0.0/13 BND XIO B3:5/10 XIO O:1.0/2 OTE O:1.0/1 EOR
%   B3:3/15  SEND_BRUSH_OUT_LTCH %
%   I:0.0/8  AUTO  "Enter Auto Mode" %
%   I:0.0/13  BRUSH_DRIVE_OUT_SS  "Hand Mode" %
%   B3:5/10  DRIVE_OUT_LS %
%   O:1.0/2  BRUSH_DRIVE_IN %
%   O:1.0/1  BRUSH_DRIVE_OUT %
% Rung: 10 %
SOR XIC B3:3/5 XIC B3:5/10 TON T4:24 1.0 3 0 EOR
%   B3:3/5  BRUSH_HAS_BEEN_IN  "Tall Bin Brush Has Been In" %
%   B3:5/10  DRIVE_OUT_LS %
%   T4:24  BRUSH_OUT_WASH_TIME  "Tall Bin Brush has been in and back out wash time" %
% Rung: 11 %
SOR XIC B3:3/4 MOV N7:38 T4:24.PRE EOR
%   B3:3/4  TALL_BIN  "TALL BIN SIZE" %
%   N7:38  TALLBIN_BRUSH_TIME  "HMI Tall Bin Brush Time" %
%   T4:24  BRUSH_OUT_WASH_TIME  "Tall Bin Brush has been in and back out wash time" %
% Rung: 12 %
% Cuts out brush time if there is a 26" bin is selected. (Removes Brush out wash timer) %
SOR XIC B3:3/3 MOV 0 T4:24.PRE EOR
%   B3:3/3  MEDIUM_BIN  "26 INCH BIN SIZE" %
%   T4:24  BRUSH_OUT_WASH_TIME  "Tall Bin Brush has been in and back out wash time" %
% Rung: 13 %
SOR MOV N7:38 T4:23.PRE EOR
%   N7:38  TALLBIN_BRUSH_TIME  "HMI Tall Bin Brush Time" %
%   T4:23  BRUSH_IN_WASH_TIME  "Tall Bin Reverse Direction" %

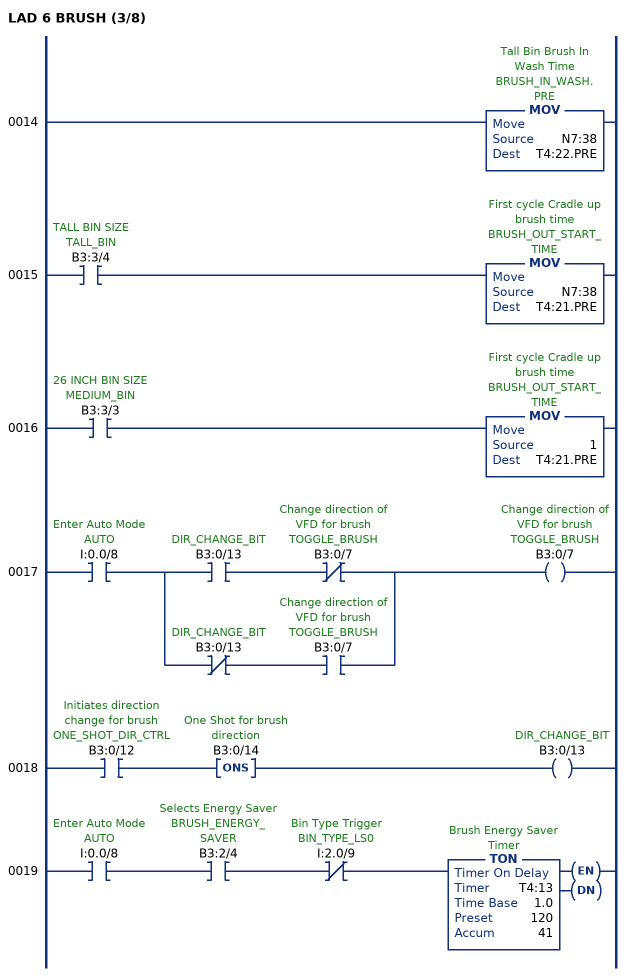
% Rung: 14 %
SOR MOV N7:38 T4:22.PRE EOR
%   N7:38  TALLBIN_BRUSH_TIME  "HMI Tall Bin Brush Time" %
%   T4:22  BRUSH_IN_WASH  "Tall Bin Brush In Wash Time" %
% Rung: 15 %
SOR XIC B3:3/4 MOV N7:38 T4:21.PRE EOR
%   B3:3/4  TALL_BIN  "TALL BIN SIZE" %
%   N7:38  TALLBIN_BRUSH_TIME  "HMI Tall Bin Brush Time" %
%   T4:21.PRE  BRUSH_OUT_START_TIME  "First cycle Cradle up brush time" %
% Rung: 16 %
SOR XIC B3:3/3 MOV 1 T4:21.PRE EOR
%   B3:3/3  MEDIUM_BIN  "26 INCH BIN SIZE" %
%   T4:21.PRE  BRUSH_OUT_START_TIME  "First cycle Cradle up brush time" %
% Rung: 17 %
SOR XIC I:0.0/8 BST XIC B3:0/13 XIO B3:0/7 NXB XIO B3:0/13 XIC B3:0/7 BND OTE B3:0/7 EOR
%   I:0.0/8  AUTO  "Enter Auto Mode" %
%   B3:0/13  DIR_CHANGE_BIT %
%   B3:0/7  TOGGLE_BRUSH  "Change direction of VFD for brush" %
% Rung: 18 %
SOR XIC B3:0/12 ONS B3:0/14 OTE B3:0/13 EOR
%   B3:0/12  ONE_SHOT_DIR_CTRL  "Initiates direction change for brush" %
%   B3:0/14  "One Shot for brush direction" %
%   B3:0/13  DIR_CHANGE_BIT %
% Rung: 19 %
SOR XIC I:0.0/8 XIC B3:2/4 XIO I:2.0/9 TON T4:13 1.0 120 41 EOR
%   I:0.0/8  AUTO  "Enter Auto Mode" %
%   B3:2/4  BRUSH_ENERGY_SAVER  "Selects Energy Saver" %
%   I:2.0/9  BIN_TYPE_LS0  "Bin Type Trigger" %
%   T4:13  "Brush Energy Saver Timer" %

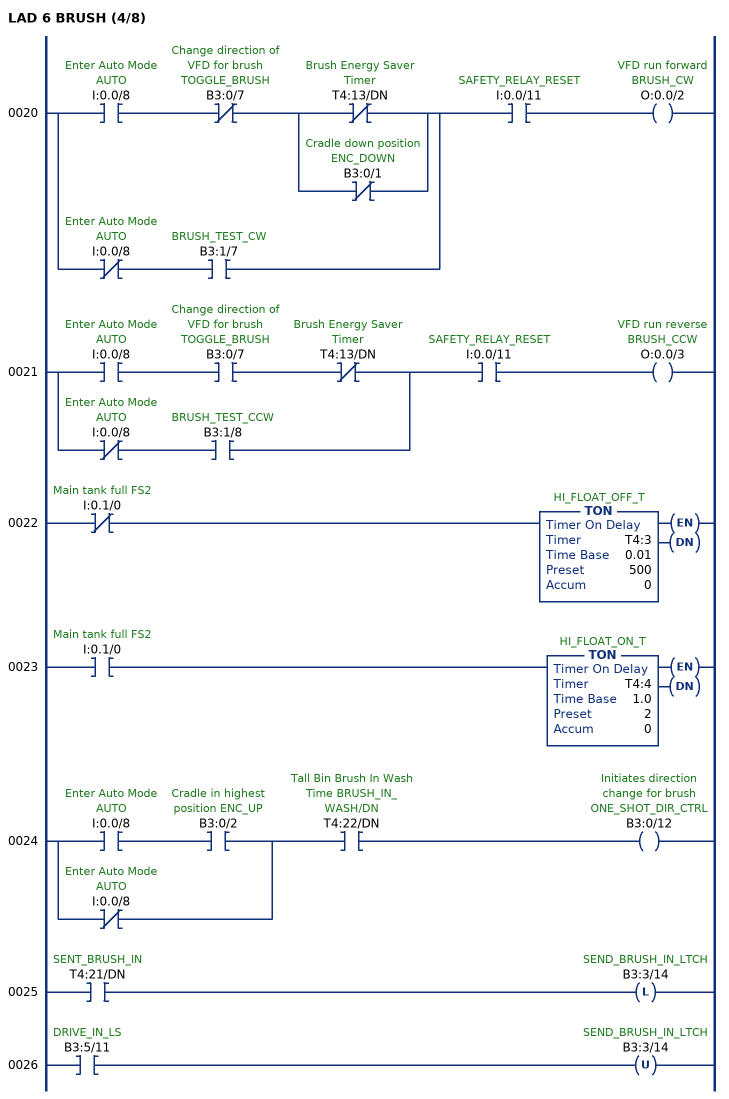
% Rung: 20 %
SOR BST XIC I:0.0/8 XIO B3:0/7 BST XIO T4:13/DN NXB XIO B3:0/1 BND NXB XIO I:0.0/8 XIC B3:1/7 BND XIC I:0.0/11 OTE O:0.0/2 EOR
%   I:0.0/8  AUTO  "Enter Auto Mode" %
%   B3:0/7  TOGGLE_BRUSH  "Change direction of VFD for brush" %
%   T4:13  "Brush Energy Saver Timer" %
%   B3:0/1  ENC_DOWN  "Cradle down position" %
%   B3:1/7  BRUSH_TEST_CW %
%   I:0.0/11  SAFETY_RELAY_RESET %
%   O:0.0/2  BRUSH_CW  "VFD run forward" %
% Rung: 21 %
SOR BST XIC I:0.0/8 XIC B3:0/7 XIO T4:13/DN NXB XIO I:0.0/8 XIC B3:1/8 BND XIC I:0.0/11 OTE O:0.0/3 EOR
%   I:0.0/8  AUTO  "Enter Auto Mode" %
%   B3:0/7  TOGGLE_BRUSH  "Change direction of VFD for brush" %
%   T4:13  "Brush Energy Saver Timer" %
%   B3:1/8  BRUSH_TEST_CCW %
%   I:0.0/11  SAFETY_RELAY_RESET %
%   O:0.0/3  BRUSH_CCW  "VFD run reverse" %
% Rung: 22 %
SOR XIO I:0.1/0 TON T4:3 0.01 500 0 EOR
%   I:0.1/0  FS2  "Main tank full" %
%   T4:3  HI_FLOAT_OFF_T %
% Rung: 23 %
SOR XIC I:0.1/0 TON T4:4 1.0 2 0 EOR
%   I:0.1/0  FS2  "Main tank full" %
%   T4:4  HI_FLOAT_ON_T %
% Rung: 24 %
SOR BST XIC I:0.0/8 XIC B3:0/2 NXB XIO I:0.0/8 BND XIC T4:22/DN OTE B3:0/12 EOR
%   I:0.0/8  AUTO  "Enter Auto Mode" %
%   B3:0/2  ENC_UP  "Cradle in highest position" %
%   T4:22  BRUSH_IN_WASH  "Tall Bin Brush In Wash Time" %
%   B3:0/12  ONE_SHOT_DIR_CTRL  "Initiates direction change for brush" %
% Rung: 25 %
SOR XIC T4:21/DN OTL B3:3/14 EOR
%   T4:21/DN  SENT_BRUSH_IN %
%   B3:3/14  SEND_BRUSH_IN_LTCH %
% Rung: 26 %
SOR XIC B3:5/11 OTU B3:3/14 EOR
%   B3:5/11  DRIVE_IN_LS %
%   B3:3/14  SEND_BRUSH_IN_LTCH %

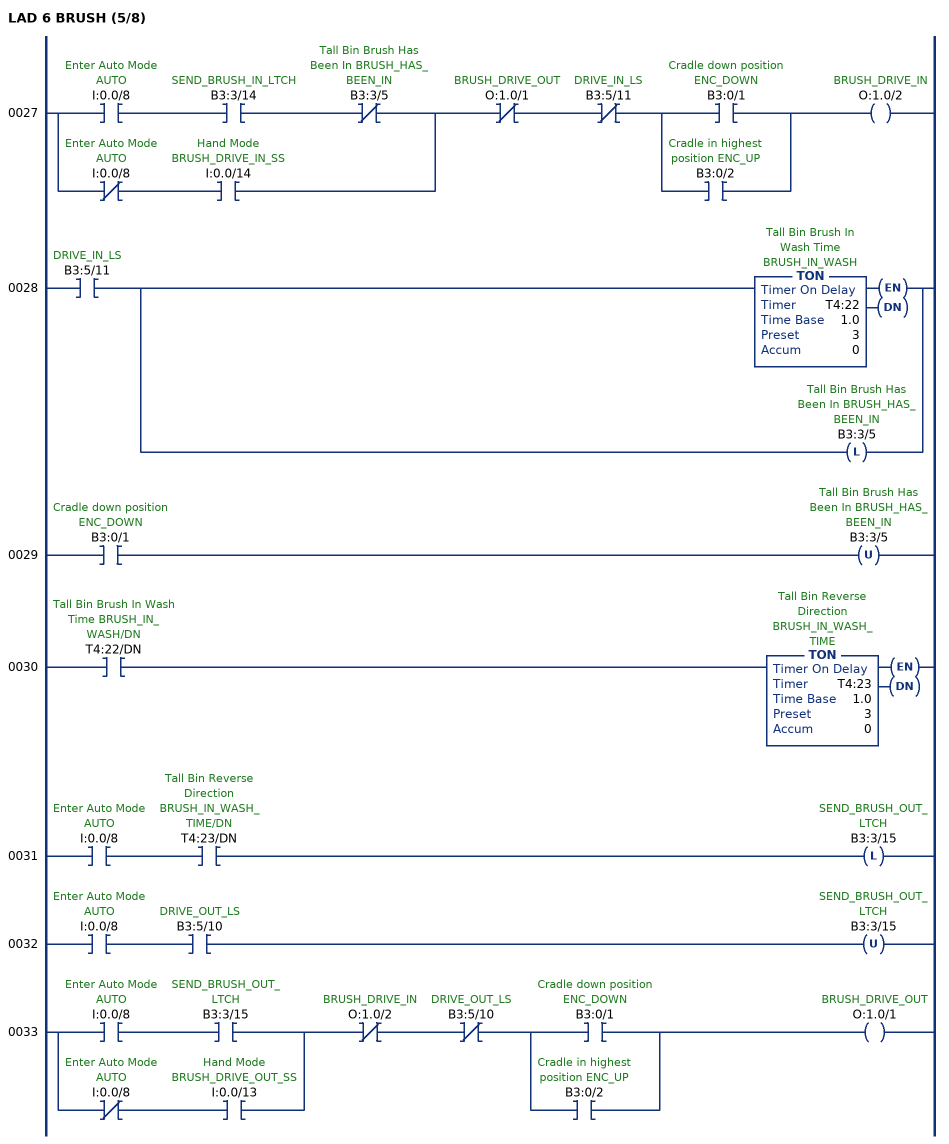
% Rung: 27 %
SOR BST XIC I:0.0/8 XIC B3:3/14 XIO B3:3/5 NXB XIO I:0.0/8 XIC I:0.0/14 BND XIO O:1.0/1 XIO B3:5/11 BST XIC B3:0/1 NXB XIC B3:0/2 BND OTE O:1.0/2 EOR
%   I:0.0/8  AUTO  "Enter Auto Mode" %
%   B3:3/14  SEND_BRUSH_IN_LTCH %
%   B3:3/5  BRUSH_HAS_BEEN_IN  "Tall Bin Brush Has Been In" %
%   I:0.0/14  BRUSH_DRIVE_IN_SS  "Hand Mode" %
%   O:1.0/1  BRUSH_DRIVE_OUT %
%   B3:5/11  DRIVE_IN_LS %
%   B3:0/1  ENC_DOWN  "Cradle down position" %
%   B3:0/2  ENC_UP  "Cradle in highest position" %
%   O:1.0/2  BRUSH_DRIVE_IN %
% Rung: 28 %
SOR XIC B3:5/11 BST TON T4:22 1.0 3 0 NXB OTL B3:3/5 BND EOR
%   B3:5/11  DRIVE_IN_LS %
%   T4:22  BRUSH_IN_WASH  "Tall Bin Brush In Wash Time" %
%   B3:3/5  BRUSH_HAS_BEEN_IN  "Tall Bin Brush Has Been In" %
% Rung: 29 %
SOR XIC B3:0/1 OTU B3:3/5 EOR
%   B3:0/1  ENC_DOWN  "Cradle down position" %
%   B3:3/5  BRUSH_HAS_BEEN_IN  "Tall Bin Brush Has Been In" %
% Rung: 30 %
SOR XIC T4:22/DN TON T4:23 1.0 3 0 EOR
%   T4:22  BRUSH_IN_WASH  "Tall Bin Brush In Wash Time" %
%   T4:23  BRUSH_IN_WASH_TIME  "Tall Bin Reverse Direction" %
% Rung: 31 %
SOR XIC I:0.0/8 XIC T4:23/DN OTL B3:3/15 EOR
%   I:0.0/8  AUTO  "Enter Auto Mode" %
%   T4:23  BRUSH_IN_WASH_TIME  "Tall Bin Reverse Direction" %
%   B3:3/15  SEND_BRUSH_OUT_LTCH %
% Rung: 32 %
SOR XIC I:0.0/8 XIC B3:5/10 OTU B3:3/15 EOR
%   I:0.0/8  AUTO  "Enter Auto Mode" %
%   B3:5/10  DRIVE_OUT_LS %
%   B3:3/15  SEND_BRUSH_OUT_LTCH %
% Rung: 33 %
SOR BST XIC I:0.0/8 XIC B3:3/15 NXB XIO I:0.0/8 XIC I:0.0/13 BND XIO O:1.0/2 XIO B3:5/10 BST XIC B3:0/1 NXB XIC B3:0/2 BND OTE O:1.0/1 EOR
%   I:0.0/8  AUTO  "Enter Auto Mode" %
%   B3:3/15  SEND_BRUSH_OUT_LTCH %
%   I:0.0/13  BRUSH_DRIVE_OUT_SS  "Hand Mode" %
%   O:1.0/2  BRUSH_DRIVE_IN %
%   B3:5/10  DRIVE_OUT_LS %
%   B3:0/1  ENC_DOWN  "Cradle down position" %
%   B3:0/2  ENC_UP  "Cradle in highest position" %
%   O:1.0/1  BRUSH_DRIVE_OUT %

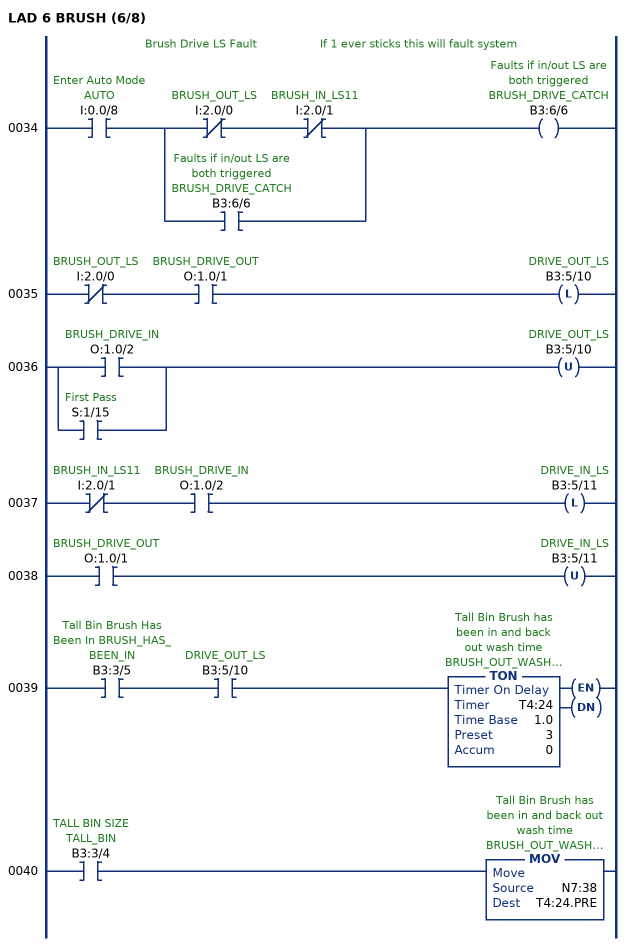
% Rung: 34 %
% Brush Drive LS Fault                  If 1 ever sticks this will fault system %
SOR XIC I:0.0/8 BST XIO I:2.0/0 XIO I:2.0/1 NXB XIC B3:6/6 BND OTE B3:6/6 EOR
%   I:0.0/8  AUTO  "Enter Auto Mode" %
%   I:2.0/0  BRUSH_OUT_LS %
%   I:2.0/1  BRUSH_IN_LS11 %
%   B3:6/6  BRUSH_DRIVE_CATCH  "Faults if in/out LS are both triggered" %
% Rung: 35 %
SOR XIO I:2.0/0 XIC O:1.0/1 OTL B3:5/10 EOR
%   I:2.0/0  BRUSH_OUT_LS %
%   O:1.0/1  BRUSH_DRIVE_OUT %
%   B3:5/10  DRIVE_OUT_LS %
% Rung: 36 %
SOR BST XIC O:1.0/2 NXB XIC S:1/15 BND OTU B3:5/10 EOR
%   O:1.0/2  BRUSH_DRIVE_IN %
%   S:1/15  "First Pass" %
%   B3:5/10  DRIVE_OUT_LS %
% Rung: 37 %
SOR XIO I:2.0/1 XIC O:1.0/2 OTL B3:5/11 EOR
%   I:2.0/1  BRUSH_IN_LS11 %
%   O:1.0/2  BRUSH_DRIVE_IN %
%   B3:5/11  DRIVE_IN_LS %
% Rung: 38 %
SOR XIC O:1.0/1 OTU B3:5/11 EOR
%   O:1.0/1  BRUSH_DRIVE_OUT %
%   B3:5/11  DRIVE_IN_LS %
% Rung: 39 %
SOR XIC B3:3/5 XIC B3:5/10 TON T4:24 1.0 3 0 EOR
%   B3:3/5  BRUSH_HAS_BEEN_IN  "Tall Bin Brush Has Been In" %
%   B3:5/10  DRIVE_OUT_LS %
%   T4:24  BRUSH_OUT_WASH_TIME  "Tall Bin Brush has been in and back out wash time" %
% Rung: 40 %
SOR XIC B3:3/4 MOV N7:38 T4:24.PRE EOR
%   B3:3/4  TALL_BIN  "TALL BIN SIZE" %
%   N7:38  TALLBIN_BRUSH_TIME  "HMI Tall Bin Brush Time" %
%   T4:24  BRUSH_OUT_WASH_TIME  "Tall Bin Brush has been in and back out wash time" %

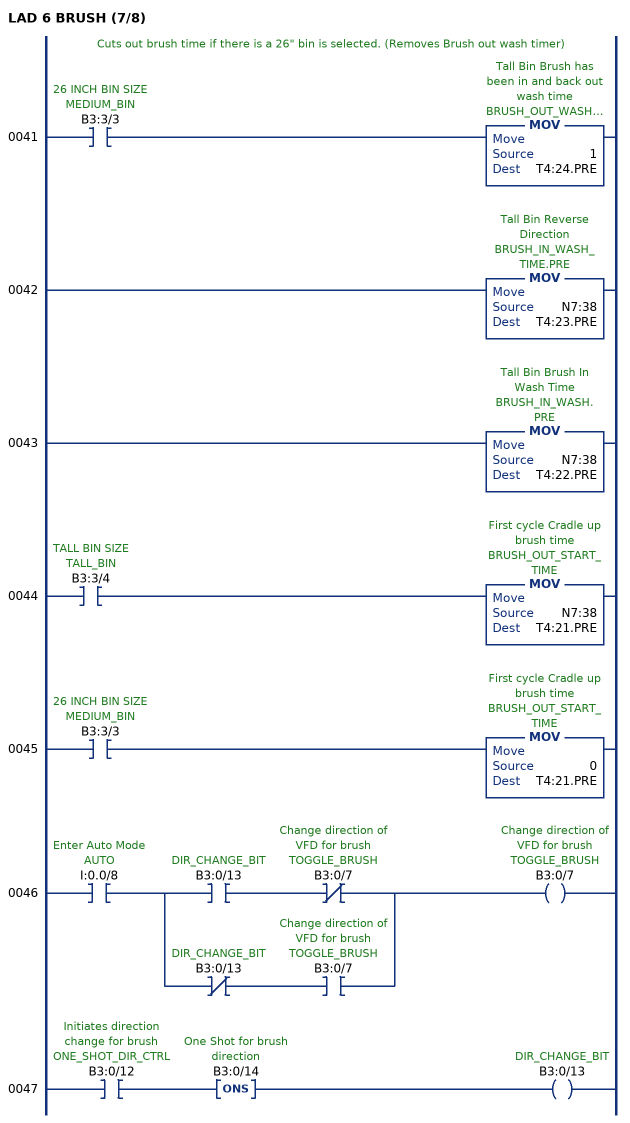
% Rung: 41 %
% Cuts out brush time if there is a 26" bin is selected. (Removes Brush out wash timer) %
SOR XIC B3:3/3 MOV 1 T4:24.PRE EOR
%   B3:3/3  MEDIUM_BIN  "26 INCH BIN SIZE" %
%   T4:24  BRUSH_OUT_WASH_TIME  "Tall Bin Brush has been in and back out wash time" %
% Rung: 42 %
SOR MOV N7:38 T4:23.PRE EOR
%   N7:38  TALLBIN_BRUSH_TIME  "HMI Tall Bin Brush Time" %
%   T4:23  BRUSH_IN_WASH_TIME  "Tall Bin Reverse Direction" %
% Rung: 43 %
SOR MOV N7:38 T4:22.PRE EOR
%   N7:38  TALLBIN_BRUSH_TIME  "HMI Tall Bin Brush Time" %
%   T4:22  BRUSH_IN_WASH  "Tall Bin Brush In Wash Time" %
% Rung: 44 %
SOR XIC B3:3/4 MOV N7:38 T4:21.PRE EOR
%   B3:3/4  TALL_BIN  "TALL BIN SIZE" %
%   N7:38  TALLBIN_BRUSH_TIME  "HMI Tall Bin Brush Time" %
%   T4:21.PRE  BRUSH_OUT_START_TIME  "First cycle Cradle up brush time" %
% Rung: 45 %
SOR XIC B3:3/3 MOV 0 T4:21.PRE EOR
%   B3:3/3  MEDIUM_BIN  "26 INCH BIN SIZE" %
%   T4:21.PRE  BRUSH_OUT_START_TIME  "First cycle Cradle up brush time" %
% Rung: 46 %
SOR XIC I:0.0/8 BST XIC B3:0/13 XIO B3:0/7 NXB XIO B3:0/13 XIC B3:0/7 BND OTE B3:0/7 EOR
%   I:0.0/8  AUTO  "Enter Auto Mode" %
%   B3:0/13  DIR_CHANGE_BIT %
%   B3:0/7  TOGGLE_BRUSH  "Change direction of VFD for brush" %
% Rung: 47 %
SOR XIC B3:0/12 ONS B3:0/14 OTE B3:0/13 EOR
%   B3:0/12  ONE_SHOT_DIR_CTRL  "Initiates direction change for brush" %
%   B3:0/14  "One Shot for brush direction" %
%   B3:0/13  DIR_CHANGE_BIT %

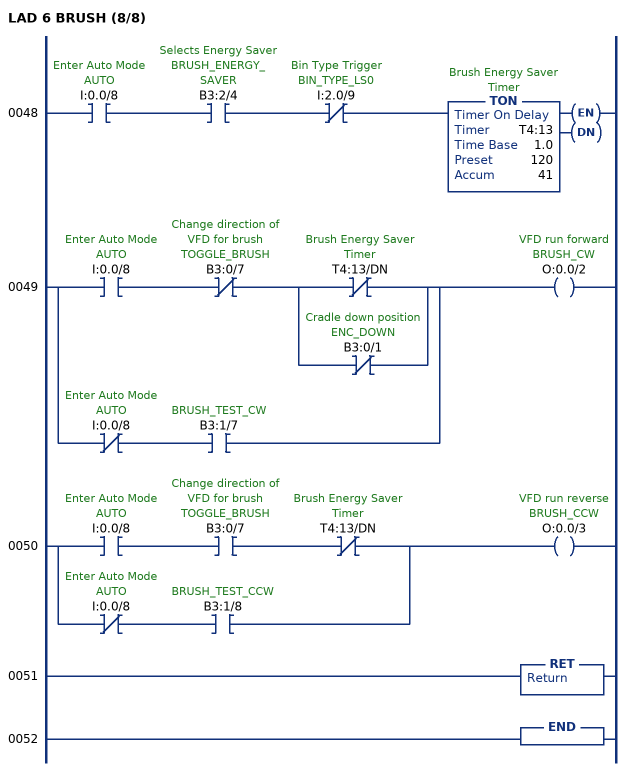
% Rung: 48 %
SOR XIC I:0.0/8 XIC B3:2/4 XIO I:2.0/9 TON T4:13 1.0 120 41 EOR
%   I:0.0/8  AUTO  "Enter Auto Mode" %
%   B3:2/4  BRUSH_ENERGY_SAVER  "Selects Energy Saver" %
%   I:2.0/9  BIN_TYPE_LS0  "Bin Type Trigger" %
%   T4:13  "Brush Energy Saver Timer" %
% Rung: 49 %
SOR BST XIC I:0.0/8 XIO B3:0/7 BST XIO T4:13/DN NXB XIO B3:0/1 BND NXB XIO I:0.0/8 XIC B3:1/7 BND OTE O:0.0/2 EOR
%   I:0.0/8  AUTO  "Enter Auto Mode" %
%   B3:0/7  TOGGLE_BRUSH  "Change direction of VFD for brush" %
%   T4:13  "Brush Energy Saver Timer" %
%   B3:0/1  ENC_DOWN  "Cradle down position" %
%   B3:1/7  BRUSH_TEST_CW %
%   O:0.0/2  BRUSH_CW  "VFD run forward" %
% Rung: 50 %
SOR BST XIC I:0.0/8 XIC B3:0/7 XIO T4:13/DN NXB XIO I:0.0/8 XIC B3:1/8 BND OTE O:0.0/3 EOR
%   I:0.0/8  AUTO  "Enter Auto Mode" %
%   B3:0/7  TOGGLE_BRUSH  "Change direction of VFD for brush" %
%   T4:13  "Brush Energy Saver Timer" %
%   B3:1/8  BRUSH_TEST_CCW %
%   O:0.0/3  BRUSH_CCW  "VFD run reverse" %
% Rung: 51 %
SOR RET EOR
% Rung: 52 %
SOR END EOR

LADDER 7 "TANK"
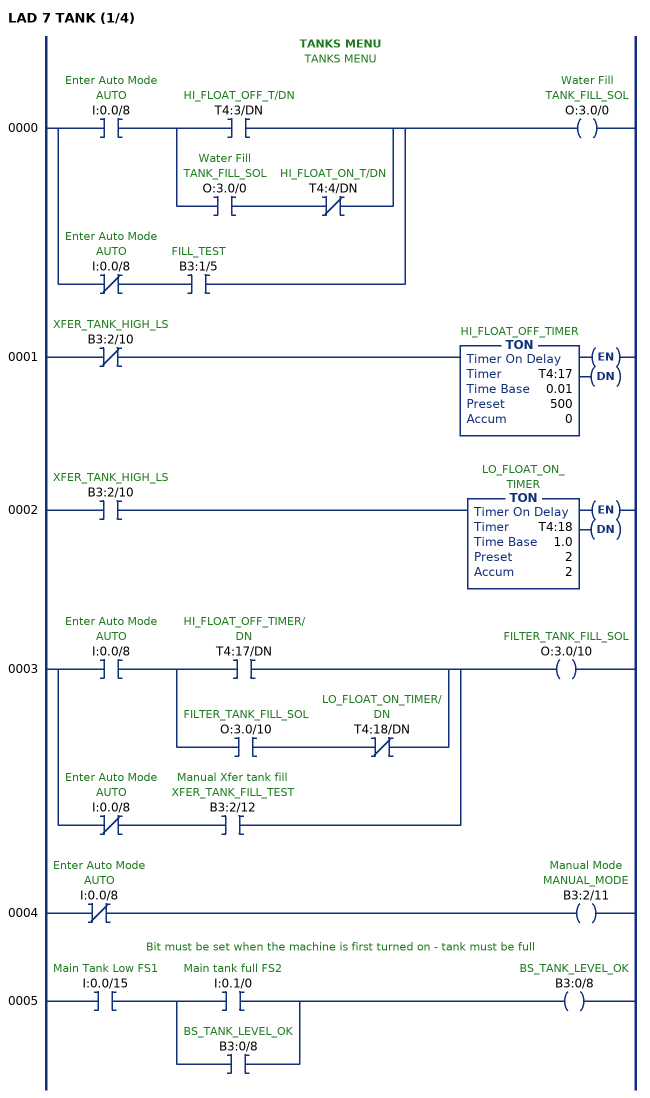
% Rung: 0 %
% TITLE: TANKS MENU %
% TANKS MENU %
SOR BST XIC I:0.0/8 BST XIC T4:3/DN NXB XIC O:3.0/0 XIO T4:4/DN BND NXB XIO I:0.0/8 XIC B3:1/5 BND OTE O:3.0/0 EOR
%   I:0.0/8  AUTO  "Enter Auto Mode" %
%   T4:3  HI_FLOAT_OFF_T %
%   O:3.0/0  TANK_FILL_SOL  "Water Fill" %
%   T4:4  HI_FLOAT_ON_T %
%   B3:1/5  FILL_TEST %
% Rung: 1 %
SOR XIO B3:2/10 TON T4:17 0.01 500 0 EOR
%   B3:2/10  XFER_TANK_HIGH_LS %
%   T4:17  HI_FLOAT_OFF_TIMER %
% Rung: 2 %
SOR XIC B3:2/10 TON T4:18 1.0 2 2 EOR
%   B3:2/10  XFER_TANK_HIGH_LS %
%   T4:18  LO_FLOAT_ON_TIMER %
% Rung: 3 %
SOR BST XIC I:0.0/8 BST XIC T4:17/DN NXB XIC O:3.0/10 XIO T4:18/DN BND NXB XIO I:0.0/8 XIC B3:2/12 BND OTE O:3.0/10 EOR
%   I:0.0/8  AUTO  "Enter Auto Mode" %
%   T4:17  HI_FLOAT_OFF_TIMER %
%   O:3.0/10  FILTER_TANK_FILL_SOL %
%   T4:18  LO_FLOAT_ON_TIMER %
%   B3:2/12  XFER_TANK_FILL_TEST  "Manual Xfer tank fill" %
% Rung: 4 %
SOR XIO I:0.0/8 OTE B3:2/11 EOR
%   I:0.0/8  AUTO  "Enter Auto Mode" %
%   B3:2/11  MANUAL_MODE  "Manual Mode" %
% Rung: 5 %
% Bit must be set when the machine is first turned on - tank must be full %
SOR XIC I:0.0/15 BST XIC I:0.1/0 NXB XIC B3:0/8 BND OTE B3:0/8 EOR
%   I:0.0/15  FS1  "Main Tank Low" %
%   I:0.1/0  FS2  "Main tank full" %
%   B3:0/8  BS_TANK_LEVEL_OK %

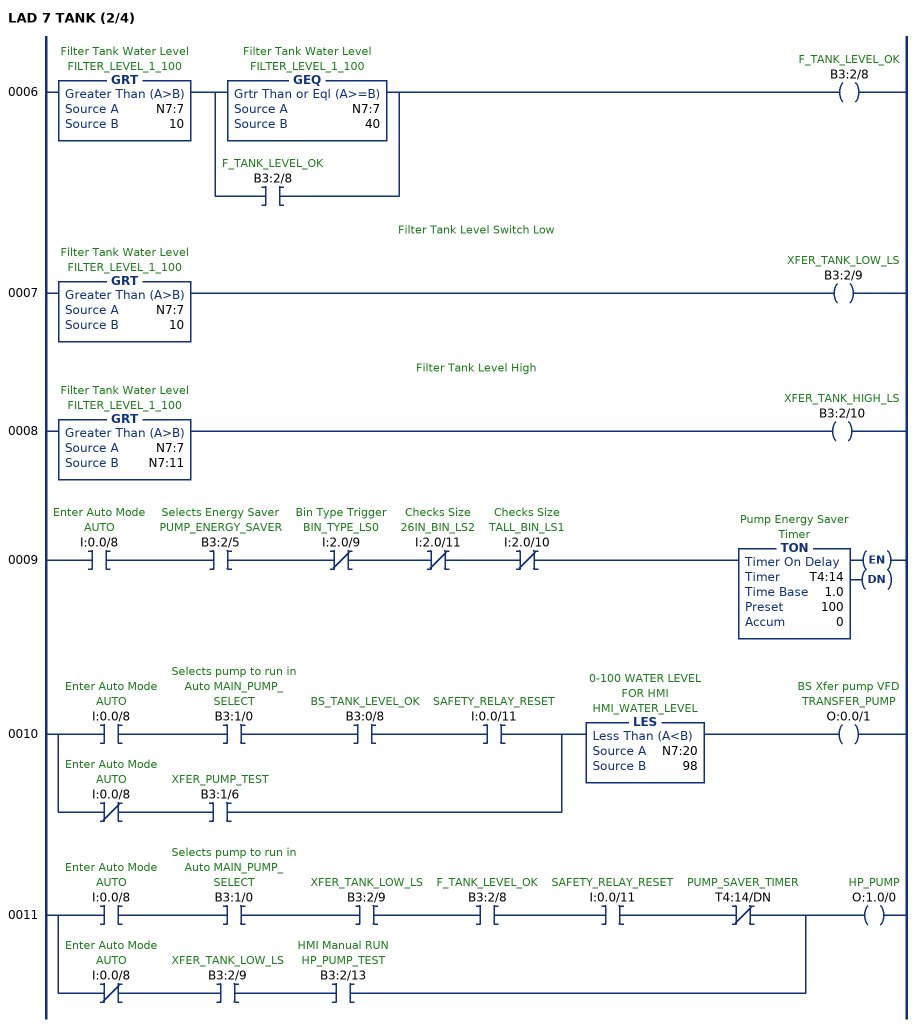
% Rung: 6 %
SOR GRT N7:7 10 BST GEQ N7:7 40 NXB XIC B3:2/8 BND OTE B3:2/8 EOR
%   N7:7  FILTER_LEVEL_1_100  "Filter Tank Water Level" %
%   B3:2/8  F_TANK_LEVEL_OK %
% Rung: 7 %
% Filter Tank Level Switch Low %
SOR GRT N7:7 10 OTE B3:2/9 EOR
%   N7:7  FILTER_LEVEL_1_100  "Filter Tank Water Level" %
%   B3:2/9  XFER_TANK_LOW_LS %
% Rung: 8 %
% Filter Tank Level High %
SOR GRT N7:7 N7:11 OTE B3:2/10 EOR
%   N7:7  FILTER_LEVEL_1_100  "Filter Tank Water Level" %
%   N7:11  FILTER_TANK_FULL_LS  "Filter Tank High Water LS" %
%   B3:2/10  XFER_TANK_HIGH_LS %
% Rung: 9 %
SOR XIC I:0.0/8 XIC B3:2/5 XIO I:2.0/9 XIO I:2.0/11 XIO I:2.0/10 TON T4:14 1.0 100 0 EOR
%   I:0.0/8  AUTO  "Enter Auto Mode" %
%   B3:2/5  PUMP_ENERGY_SAVER  "Selects Energy Saver" %
%   I:2.0/9  BIN_TYPE_LS0  "Bin Type Trigger" %
%   I:2.0/11  26IN_BIN_LS2  "Checks Size" %
%   I:2.0/10  TALL_BIN_LS1  "Checks Size" %
%   T4:14  "Pump Energy Saver Timer" %
% Rung: 10 %
SOR BST XIC I:0.0/8 XIC B3:1/0 XIC B3:0/8 XIC I:0.0/11 NXB XIO I:0.0/8 XIC B3:1/6 BND LES N7:20 98 OTE O:0.0/1 EOR
%   I:0.0/8  AUTO  "Enter Auto Mode" %
%   B3:1/0  MAIN_PUMP_SELECT  "Selects pump to run in Auto" %
%   B3:0/8  BS_TANK_LEVEL_OK %
%   I:0.0/11  SAFETY_RELAY_RESET %
%   B3:1/6  XFER_PUMP_TEST %
%   N7:20  HMI_WATER_LEVEL  "0-100 WATER LEVEL FOR HMI" %
%   O:0.0/1  TRANSFER_PUMP  "BS Xfer pump VFD" %
% Rung: 11 %
SOR BST XIC I:0.0/8 XIC B3:1/0 XIC B3:2/9 XIC B3:2/8 XIC I:0.0/11 XIO T4:14/DN NXB XIO I:0.0/8 XIC B3:2/9 XIC B3:2/13 BND OTE O:1.0/0 EOR
%   I:0.0/8  AUTO  "Enter Auto Mode" %
%   B3:1/0  MAIN_PUMP_SELECT  "Selects pump to run in Auto" %
%   B3:2/9  XFER_TANK_LOW_LS %
%   B3:2/8  F_TANK_LEVEL_OK %
%   I:0.0/11  SAFETY_RELAY_RESET %
%   T4:14/DN  PUMP_SAVER_TIMER %
%   B3:2/13  HP_PUMP_TEST  "HMI Manual RUN" %
%   O:1.0/0  HP_PUMP %

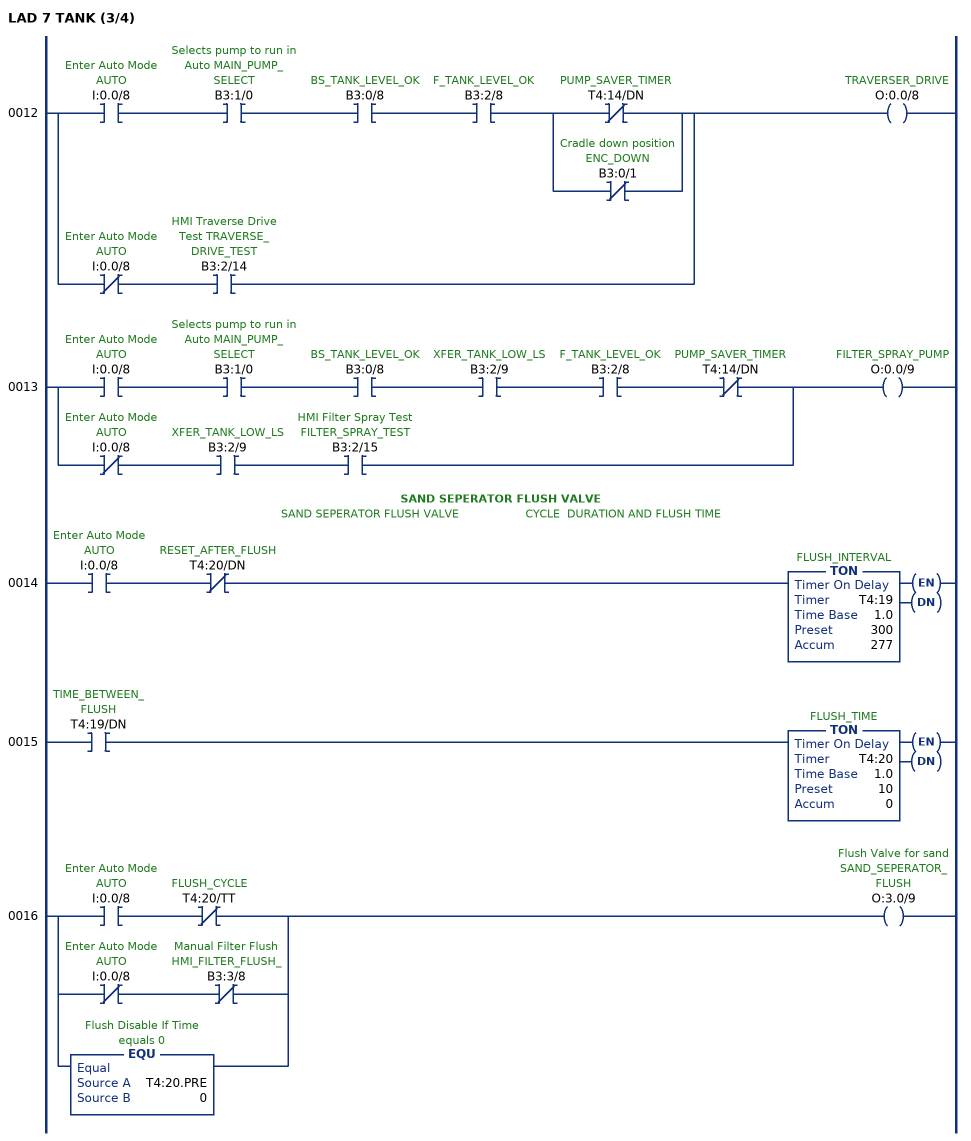
% Rung: 12 %
SOR BST XIC I:0.0/8 XIC B3:1/0 XIC B3:0/8 XIC B3:2/8 BST XIO T4:14/DN NXB XIO B3:0/1 BND NXB XIO I:0.0/8 XIC B3:2/14 BND OTE O:0.0/8 EOR
%   I:0.0/8  AUTO  "Enter Auto Mode" %
%   B3:1/0  MAIN_PUMP_SELECT  "Selects pump to run in Auto" %
%   B3:0/8  BS_TANK_LEVEL_OK %
%   B3:2/8  F_TANK_LEVEL_OK %
%   T4:14/DN  PUMP_SAVER_TIMER %
%   B3:0/1  ENC_DOWN  "Cradle down position" %
%   B3:2/14  TRAVERSE_DRIVE_TEST  "HMI Traverse Drive Test" %
%   O:0.0/8  TRAVERSER_DRIVE %
% Rung: 13 %
SOR BST XIC I:0.0/8 XIC B3:1/0 XIC B3:0/8 XIC B3:2/9 XIC B3:2/8 XIO T4:14/DN NXB XIO I:0.0/8 XIC B3:2/9 XIC B3:2/15 BND OTE O:0.0/9 EOR
%   I:0.0/8  AUTO  "Enter Auto Mode" %
%   B3:1/0  MAIN_PUMP_SELECT  "Selects pump to run in Auto" %
%   B3:0/8  BS_TANK_LEVEL_OK %
%   B3:2/9  XFER_TANK_LOW_LS %
%   B3:2/8  F_TANK_LEVEL_OK %
%   T4:14/DN  PUMP_SAVER_TIMER %
%   B3:2/15  FILTER_SPRAY_TEST  "HMI Filter Spray Test" %
%   O:0.0/9  FILTER_SPRAY_PUMP %
% Rung: 14 %
% TITLE: SAND SEPERATOR FLUSH VALVE %
% SAND SEPERATOR FLUSH VALVE                   CYCLE  DURATION AND FLUSH TIME %
SOR XIC I:0.0/8 XIO T4:20/DN TON T4:19 1.0 300 277 EOR
%   I:0.0/8  AUTO  "Enter Auto Mode" %
%   T4:20/DN  RESET_AFTER_FLUSH %
%   T4:19  FLUSH_INTERVAL %
% Rung: 15 %
SOR XIC T4:19/DN TON T4:20 1.0 10 0 EOR
%   T4:19/DN  TIME_BETWEEN_FLUSH %
%   T4:20  FLUSH_TIME %
% Rung: 16 %
SOR BST XIC I:0.0/8 XIO T4:20/TT NXB BST XIO I:0.0/8 XIO B3:3/8 NXB EQU T4:20.PRE 0 BND BND OTE O:3.0/9 EOR
%   I:0.0/8  AUTO  "Enter Auto Mode" %
%   T4:20/TT  FLUSH_CYCLE %
%   B3:3/8  HMI_FILTER_FLUSH_  "Manual Filter Flush" %
%   T4:20.PRE  "Flush Disable If Time equals 0" %
%   O:3.0/9  SAND_SEPERATOR_FLUSH  "Flush Valve for sand" %

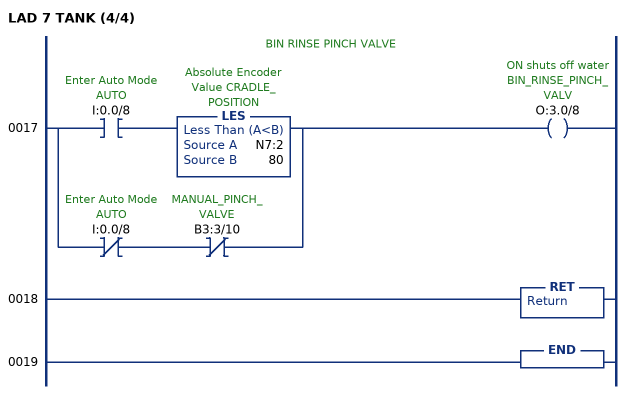
% Rung: 17 %
% BIN RINSE PINCH VALVE %
SOR BST XIC I:0.0/8 LES N7:2 80 NXB XIO I:0.0/8 XIO B3:3/10 BND OTE O:3.0/8 EOR
%   I:0.0/8  AUTO  "Enter Auto Mode" %
%   N7:2  CRADLE_POSITION  "Absolute Encoder Value" %
%   B3:3/10  MANUAL_PINCH_VALVE %
%   O:3.0/8  BIN_RINSE_PINCH_VALV  "ON shuts off water" %
% Rung: 18 %
SOR RET EOR
% Rung: 19 %
SOR END EOR

LADDER 8 "AUXILARY"
